REGION Network 16: 100 - return - wait for handshake with other instances
   RUNG wire#powerrail
      { S7_Templates := "SrcType := Int" } EQ_Contact(in1 := #cnt, in2 := 100)
      wire#w1
      Move(in := 0.0, out1 => #HydraulicCylinder.PressureCmd)
      Move(in := 0.0, out1 => #HydraulicCylinder.FlowCmd)
   END_RUNG
   RUNG wire#w1
      R_Coil( #dataDigiforce.Start )
   END_RUNG
   RUNG wire#w1
      Coil( #dataFitting.Returning )
   END_RUNG
   RUNG wire#w1
      Contact( #dataFitting.ContinueReturn )
      Move(in := 105, out1 => #cnt)
   END_RUNG
   // the same network as SCL:
   #_w1 := #cnt = 100;
   IF #_w1 THEN
       #HydraulicCylinder.PressureCmd := 0.0;
       #HydraulicCylinder.FlowCmd := 0.0;
       #dataDigiforce.Start := FALSE;
   END_IF;
   #dataFitting.Returning := #_w1;
   IF #_w1 AND #dataFitting.ContinueReturn THEN #cnt := 105; END_IF;
END_REGION

REGION Network 17: 105 - Start returning
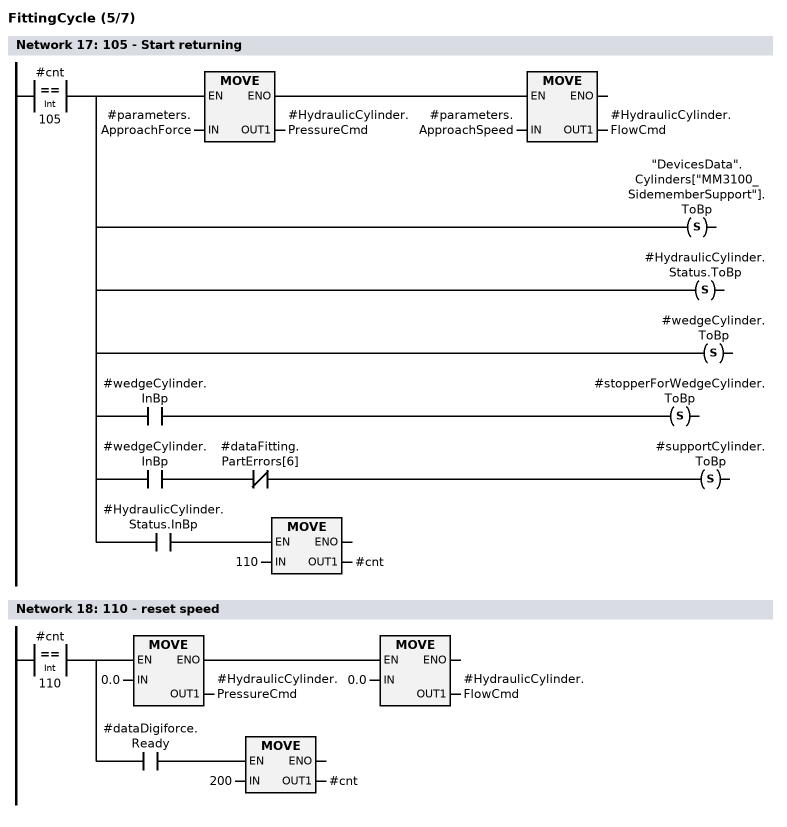
   RUNG wire#powerrail
      { S7_Templates := "SrcType := Int" } EQ_Contact(in1 := #cnt, in2 := 105)
      wire#w1
      Move(in := #parameters.ApproachForce, out1 => #HydraulicCylinder.PressureCmd)
      Move(in := #parameters.ApproachSpeed, out1 => #HydraulicCylinder.FlowCmd)
   END_RUNG
   RUNG wire#w1
      S_Coil( "DevicesData".Cylinders["MM3100_SidememberSupport"].ToBp )
   END_RUNG
   RUNG wire#w1
      S_Coil( #HydraulicCylinder.Status.ToBp )
   END_RUNG
   RUNG wire#w1
      S_Coil( #wedgeCylinder.ToBp )
   END_RUNG
   RUNG wire#w1
      Contact( #wedgeCylinder.InBp )
      S_Coil( #stopperForWedgeCylinder.ToBp )
   END_RUNG
   RUNG wire#w1
      Contact( #wedgeCylinder.InBp )
      I_Contact( #dataFitting.PartErrors[6] )
      S_Coil( #supportCylinder.ToBp )
   END_RUNG
   RUNG wire#w1
      Contact( #HydraulicCylinder.Status.InBp )
      Move(in := 110, out1 => #cnt)
   END_RUNG
   // the same network as SCL:
   #_w1 := #cnt = 105;
   IF #_w1 THEN
       #HydraulicCylinder.PressureCmd := #parameters.ApproachForce;
       #HydraulicCylinder.FlowCmd := #parameters.ApproachSpeed;
       "DevicesData".Cylinders["MM3100_SidememberSupport"].ToBp := TRUE;
       #HydraulicCylinder.Status.ToBp := TRUE;
       #wedgeCylinder.ToBp := TRUE;
   END_IF;
   IF #_w1 AND #wedgeCylinder.InBp THEN #stopperForWedgeCylinder.ToBp := TRUE; END_IF;
   IF #_w1 AND #wedgeCylinder.InBp AND NOT #dataFitting.PartErrors[6] THEN
       #supportCylinder.ToBp := TRUE;
   END_IF;
   IF #_w1 AND #HydraulicCylinder.Status.InBp THEN #cnt := 110; END_IF;
END_REGION

REGION Network 18: 110 - reset speed
   RUNG wire#powerrail
      { S7_Templates := "SrcType := Int" } EQ_Contact(in1 := #cnt, in2 := 110)
      wire#w1
      Move(in := 0.0, out1 => #HydraulicCylinder.PressureCmd)
      Move(in := 0.0, out1 => #HydraulicCylinder.FlowCmd)
   END_RUNG
   RUNG wire#w1
      Contact( #dataDigiforce.Ready )
      Move(in := 200, out1 => #cnt)
   END_RUNG
   // the same network as SCL:
   #_w1 := #cnt = 110;
   IF #_w1 THEN
       #HydraulicCylinder.PressureCmd := 0.0;
       #HydraulicCylinder.FlowCmd := 0.0;
   END_IF;
   IF #_w1 AND #dataDigiforce.Ready THEN #cnt := 200; END_IF;
END_REGION

REGION Network 19: 200 - Move all cylinders to basic - evaluate result
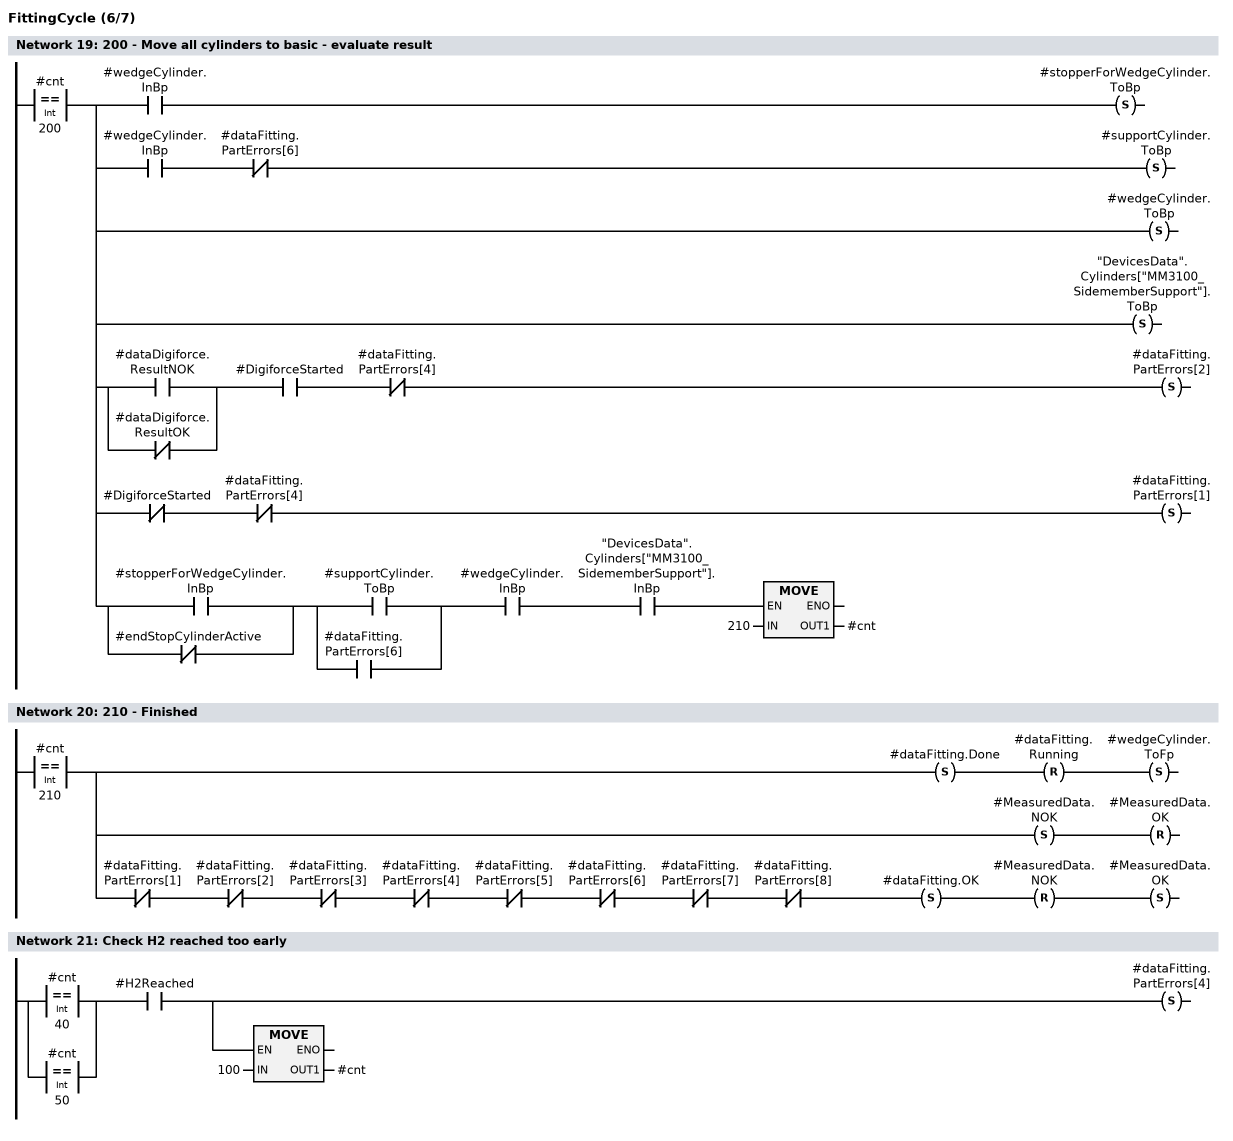
   RUNG wire#powerrail
      { S7_Templates := "SrcType := Int" } EQ_Contact(in1 := #cnt, in2 := 200)
      wire#w1
      Contact( #wedgeCylinder.InBp )
      S_Coil( #stopperForWedgeCylinder.ToBp )
   END_RUNG
   RUNG wire#w1
      Contact( #wedgeCylinder.InBp )
      I_Contact( #dataFitting.PartErrors[6] )
      S_Coil( #supportCylinder.ToBp )
   END_RUNG
   RUNG wire#w1
      S_Coil( #wedgeCylinder.ToBp )
   END_RUNG
   RUNG wire#w1
      S_Coil( "DevicesData".Cylinders["MM3100_SidememberSupport"].ToBp )
   END_RUNG
   RUNG wire#w1
      Contact( #dataDigiforce.ResultNOK )
      wire#w2
      Contact( #DigiforceStarted )
      I_Contact( #dataFitting.PartErrors[4] )
      S_Coil( #dataFitting.PartErrors[2] )
   END_RUNG
   RUNG wire#w1
      I_Contact( #dataDigiforce.ResultOK )
   END_RUNG wire#w2
   RUNG wire#w1
      I_Contact( #DigiforceStarted )
      I_Contact( #dataFitting.PartErrors[4] )
      S_Coil( #dataFitting.PartErrors[1] )
   END_RUNG
   RUNG wire#w1
      Contact( #stopperForWedgeCylinder.InBp )
      wire#w3
      Contact( #supportCylinder.ToBp )
      wire#w4
      Contact( #wedgeCylinder.InBp )
      Contact( "DevicesData".Cylinders["MM3100_SidememberSupport"].InBp )
      Move(in := 210, out1 => #cnt)
   END_RUNG
   RUNG wire#w1
      I_Contact( #endStopCylinderActive )
   END_RUNG wire#w3
   RUNG wire#w3
      Contact( #dataFitting.PartErrors[6] )
   END_RUNG wire#w4
   // the same network as SCL:
   #_w1 := #cnt = 200;
   IF #_w1 AND #wedgeCylinder.InBp THEN #stopperForWedgeCylinder.ToBp := TRUE; END_IF;
   IF #_w1 AND #wedgeCylinder.InBp AND NOT #dataFitting.PartErrors[6] THEN
       #supportCylinder.ToBp := TRUE;
   END_IF;
   IF #_w1 THEN
       #wedgeCylinder.ToBp := TRUE;
       "DevicesData".Cylinders["MM3100_SidememberSupport"].ToBp := TRUE;
   END_IF;
   IF #_w1 AND (#dataDigiforce.ResultNOK OR NOT #dataDigiforce.ResultOK) AND #DigiforceStarted AND NOT #dataFitting.PartErrors[4] THEN
       #dataFitting.PartErrors[2] := TRUE;
   END_IF;
   IF #_w1 AND NOT #DigiforceStarted AND NOT #dataFitting.PartErrors[4] THEN
       #dataFitting.PartErrors[1] := TRUE;
   END_IF;
   IF #_w1 AND (#stopperForWedgeCylinder.InBp OR NOT #endStopCylinderActive) AND (#supportCylinder.ToBp OR #dataFitting.PartErrors[6]) AND #wedgeCylinder.InBp AND "DevicesData".Cylinders["MM3100_SidememberSupport"].InBp THEN
       #cnt := 210;
   END_IF;
END_REGION

REGION Network 20: 210 - Finished
   RUNG wire#powerrail
      { S7_Templates := "SrcType := Int" } EQ_Contact(in1 := #cnt, in2 := 210)
      wire#w1
      S_Coil( #dataFitting.Done )
      R_Coil( #dataFitting.Running )
      S_Coil( #wedgeCylinder.ToFp )
   END_RUNG
   RUNG wire#w1
      S_Coil( #MeasuredData.NOK )
      R_Coil( #MeasuredData.OK )
   END_RUNG
   RUNG wire#w1
      I_Contact( #dataFitting.PartErrors[1] )
      I_Contact( #dataFitting.PartErrors[2] )
      I_Contact( #dataFitting.PartErrors[3] )
      I_Contact( #dataFitting.PartErrors[4] )
      I_Contact( #dataFitting.PartErrors[5] )
      I_Contact( #dataFitting.PartErrors[6] )
      I_Contact( #dataFitting.PartErrors[7] )
      I_Contact( #dataFitting.PartErrors[8] )
      S_Coil( #dataFitting.OK )
      R_Coil( #MeasuredData.NOK )
      S_Coil( #MeasuredData.OK )
   END_RUNG
   // the same network as SCL:
   #_w1 := #cnt = 210;
   IF #_w1 THEN
       #dataFitting.Done := TRUE;
       #dataFitting.Running := FALSE;
       #wedgeCylinder.ToFp := TRUE;
       #MeasuredData.NOK := TRUE;
       #MeasuredData.OK := FALSE;
   END_IF;
   IF #_w1 AND NOT #dataFitting.PartErrors[1] AND NOT #dataFitting.PartErrors[2] AND NOT #dataFitting.PartErrors[3] AND NOT #dataFitting.PartErrors[4] AND NOT #dataFitting.PartErrors[5] AND NOT #dataFitting.PartErrors[6] AND NOT #dataFitting.PartErrors[7] AND NOT #dataFitting.PartErrors[8] THEN
       #dataFitting.OK := TRUE;
       #MeasuredData.NOK := FALSE;
       #MeasuredData.OK := TRUE;
   END_IF;
END_REGION

REGION Network 21: Check H2 reached too early
   RUNG wire#powerrail
      { S7_Templates := "SrcType := Int" } EQ_Contact(in1 := #cnt, in2 := 40)
      wire#w1
      Contact( #H2Reached )
      wire#w2
      S_Coil( #dataFitting.PartErrors[4] )
   END_RUNG
   RUNG wire#powerrail
      { S7_Templates := "SrcType := Int" } EQ_Contact(in1 := #cnt, in2 := 50)
   END_RUNG wire#w1
   RUNG wire#w2
      Move(in := 100, out1 => #cnt)
   END_RUNG
   // the same network as SCL:
   IF ((#cnt = 40) OR (#cnt = 50)) AND #H2Reached THEN
       #dataFitting.PartErrors[4] := TRUE;
       #cnt := 100;
   END_IF;
END_REGION

REGION Network 22: Timeout
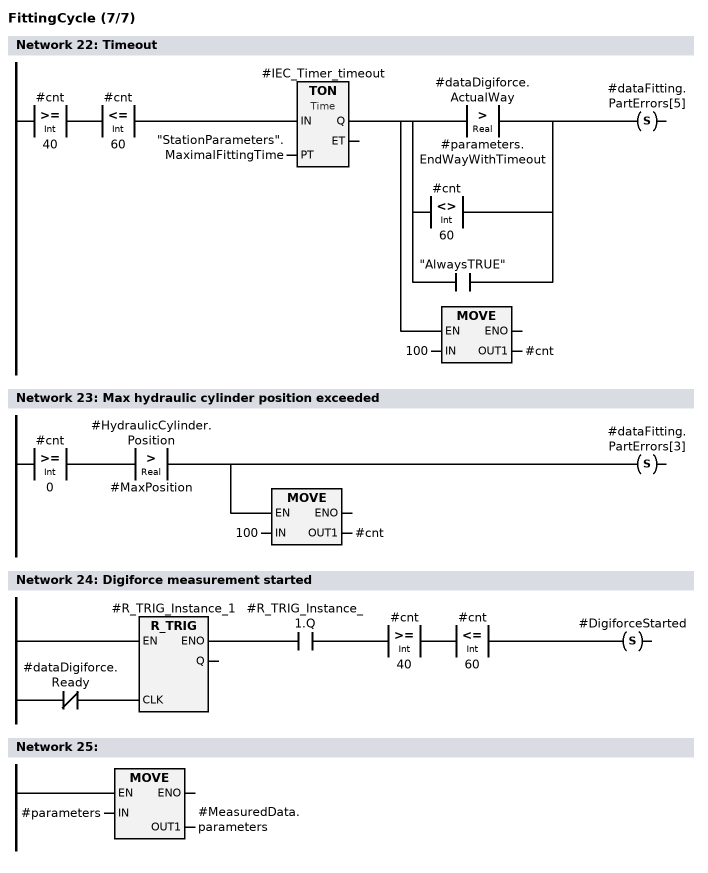
   RUNG wire#powerrail
      { S7_Templates := "SrcType := Int" } GE_Contact(in1 := #cnt, in2 := 40)
      { S7_Templates := "SrcType := Int" } LE_Contact(in1 := #cnt, in2 := 60)
      { S7_Templates := "time_type := Time" } #IEC_Timer_timeout.TON(pt := "StationParameters".MaximalFittingTime, et =>)
      wire#w1
      { S7_Templates := "SrcType := Real" } GT_Contact(in1 := #dataDigiforce.ActualWay, in2 := #parameters.EndWayWithTimeout)
      wire#w2
      S_Coil( #dataFitting.PartErrors[5] )
   END_RUNG
   RUNG wire#w1
      { S7_Templates := "SrcType := Int" } NE_Contact(in1 := #cnt, in2 := 60)
   END_RUNG wire#w2
   RUNG wire#w1
      Contact( "AlwaysTRUE" )
   END_RUNG wire#w2
   RUNG wire#w1
      Move(in := 100, out1 => #cnt)
   END_RUNG
   // the same network as SCL:
   #IEC_Timer_timeout(IN := (#cnt >= 40) AND (#cnt <= 60), PT := "StationParameters".MaximalFittingTime);   // TON
   IF #IEC_Timer_timeout.Q AND ((#dataDigiforce.ActualWay > #parameters.EndWayWithTimeout) OR (#cnt <> 60) OR "AlwaysTRUE") THEN
       #dataFitting.PartErrors[5] := TRUE;
   END_IF;
   IF #IEC_Timer_timeout.Q THEN #cnt := 100; END_IF;
END_REGION

REGION Network 23: Max hydraulic cylinder position exceeded
   RUNG wire#powerrail
      { S7_Templates := "SrcType := Int" } GE_Contact(in1 := #cnt, in2 := 0)
      { S7_Templates := "SrcType := Real" } GT_Contact(in1 := #HydraulicCylinder.Position, in2 := #MaxPosition)
      wire#w1
      S_Coil( #dataFitting.PartErrors[3] )
   END_RUNG
   RUNG wire#w1
      Move(in := 100, out1 => #cnt)
   END_RUNG
   // the same network as SCL:
   IF (#cnt >= 0) AND (#HydraulicCylinder.Position > #MaxPosition) THEN
       #dataFitting.PartErrors[3] := TRUE;
       #cnt := 100;
   END_IF;
END_REGION

REGION Network 24: Digiforce measurement started
   RUNG wire#powerrail
      #R_TRIG_Instance_1.R_TRIG(CLK := wire#w1, Q =>)
      Contact( #R_TRIG_Instance_1.Q )
      { S7_Templates := "SrcType := Int" } GE_Contact(in1 := #cnt, in2 := 40)
      { S7_Templates := "SrcType := Int" } LE_Contact(in1 := #cnt, in2 := 60)
      S_Coil( #DigiforceStarted )
   END_RUNG
   RUNG wire#powerrail
      I_Contact( #dataDigiforce.Ready )
   END_RUNG wire#w1
   // the same network as SCL:
   #R_TRIG_Instance_1(CLK := NOT #dataDigiforce.Ready, ENO => #_w1);   // R_TRIG
   IF #_w1 AND #R_TRIG_Instance_1.Q AND (#cnt >= 40) AND (#cnt <= 60) THEN #DigiforceStarted := TRUE; END_IF;
END_REGION

REGION Network 25
   RUNG wire#powerrail
      Move(in := #parameters, out1 => #MeasuredData.parameters)
   END_RUNG
   // the same network as SCL:
   #MeasuredData.parameters := #parameters;
END_REGION
END_FUNCTION_BLOCK

FUNCTION_BLOCK "HydraulicCylinder"   // FB17, LAD
{ S7_Optimized_Access := 'TRUE' }
VERSION : 0.1
// stored: AutoNumber true, IsIECCheckEnabled false, IsRetainMemResEnabled false, MemoryReserve 100, SetENOAutomatically false, UDAEnableTagReadback false
   VAR_INPUT
      HydraulicActive : Bool;
      BasicPositionMin : Real;
      BasicPositionMax : Real;
      MaxPosition : Real;
      ManualCommand : Int;
      CylinderNumber : Int;
   END_VAR
   VAR_IN_OUT
      data : "UDT_HydraulicCylinderData";
   END_VAR
   VAR
      dataOld : "UDT_HydraulicCylinderData";
      noCollision { S7_SetPoint := 'True'} : Bool;
      IEC_Timer_0_Instance { S7_SetPoint := 'True'} : TON_TIME;
      R_TRIG_Instance { S7_SetPoint := 'True'} : R_TRIG;
      difference { S7_SetPoint := 'True'} : Real;
      re : Real;
      IEC_Timer_0_Instance_1 { S7_SetPoint := 'True'} : TON_TIME;
      RampFunction_Instance { S7_SetPoint := 'True'} : RampFunction;
      BasicPositionMin_1mm_margin : Real;
      BasicPositionMax_1mm_margin : Real;
   END_VAR
   VAR_TEMP
      command : Int;
   END_VAR
   VAR_TEMP   // added for the SCL form of the ladder/FBD networks
      _w1 : Bool;
   END_VAR
BEGIN

REGION Network 1
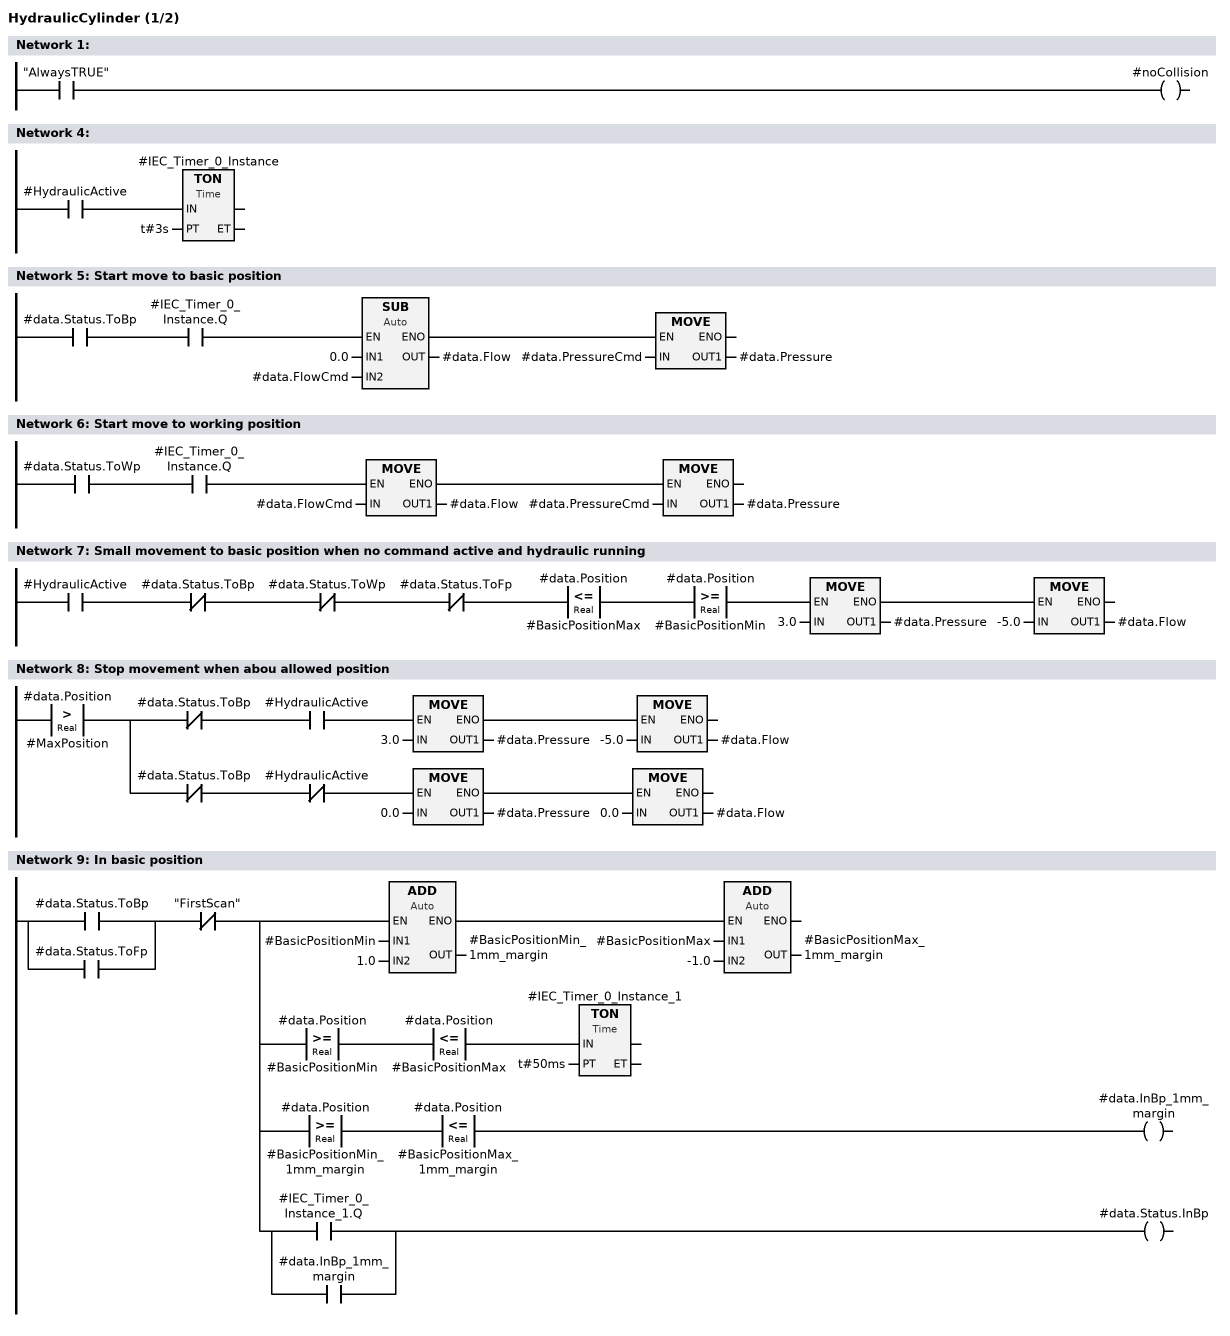
   RUNG wire#powerrail
      Contact( "AlwaysTRUE" )
      Coil( #noCollision )
   END_RUNG
   // the same network as SCL:
   #noCollision := "AlwaysTRUE";
END_REGION

REGION Network 2 (SCL)
   #command := #ManualCommand - #CylinderNumber;

   IF #command > 100 THEN
       "SandBoxData".MnualCommandMem := #command;
   END_IF;
   IF #command = 5000 THEN
       #data.Status.ToBp := true;
   END_IF;
   IF #command = 6000 THEN
       #data.Status.ToWp := true;
   END_IF;
   IF #command = 7000 THEN
       #data.Status.ToFp := true;
   END_IF;
END_REGION

REGION Network 3 (SCL): check new cylinder command
   //check if basic position req movement changed
   IF #data.Status.ToBp <> #dataOld.Status.ToBp AND #data.Status.ToBp THEN
       #data.Status.ToFp := false;
       #data.Status.ToWp := false;
       IF #noCollision THEN
           #data.Status.ToFp := false;
           #data.Status.ToWp := false;
       ELSE
           #data.Status.ToBp := false;
       END_IF;
   END_IF;
   //check if work position req movement changed
   IF #data.Status.ToWp <> #dataOld.Status.ToWp AND #data.Status.ToWp THEN
       IF #noCollision  THEN
           #data.Status.ToFp := false;
           #data.Status.ToBp := false;
       ELSE
           #data.Status.ToWp := false;
       END_IF;
   END_IF;
   //check if free position req movement changed
   IF #data.Status.ToFp <> #dataOld.Status.ToFp AND #data.Status.ToFp THEN
       #data.Status.ToBp := false;
       #data.Status.ToWp := false;
       IF #noCollision THEN
           #data.Status.ToBp := false;
           #data.Status.ToWp := false;
       ELSE
           #data.Status.ToFp := false;
       END_IF;
   END_IF;
   //store actual cylinder status to old
   #dataOld.Status := #data.Status;
END_REGION

REGION Network 4
   RUNG wire#powerrail
      Contact( #HydraulicActive )
      { S7_Templates := "time_type := Time" } #IEC_Timer_0_Instance.TON(pt := t#3s, et =>)
   END_RUNG
   // the same network as SCL:
   #IEC_Timer_0_Instance(IN := #HydraulicActive, PT := t#3s);   // TON
END_REGION

REGION Network 5: Start move to basic position
   RUNG wire#powerrail
      Contact( #data.Status.ToBp )
      Contact( #IEC_Timer_0_Instance.Q )
      Sub(in1 := 0.0, in2 := #data.FlowCmd, out => #data.Flow)
      Move(in := #data.PressureCmd, out1 => #data.Pressure)
   END_RUNG
   // the same network as SCL:
   IF #data.Status.ToBp AND #IEC_Timer_0_Instance.Q THEN
       #data.Flow := 0.0 - #data.FlowCmd;
       #data.Pressure := #data.PressureCmd;
   END_IF;
END_REGION

REGION Network 6: Start move to working position
   RUNG wire#powerrail
      Contact( #data.Status.ToWp )
      Contact( #IEC_Timer_0_Instance.Q )
      Move(in := #data.FlowCmd, out1 => #data.Flow)
      Move(in := #data.PressureCmd, out1 => #data.Pressure)
   END_RUNG
   // the same network as SCL:
   IF #data.Status.ToWp AND #IEC_Timer_0_Instance.Q THEN
       #data.Flow := #data.FlowCmd;
       #data.Pressure := #data.PressureCmd;
   END_IF;
END_REGION

REGION Network 7: Small movement to basic position when no command active and hydraulic running
   RUNG wire#powerrail
      Contact( #HydraulicActive )
      I_Contact( #data.Status.ToBp )
      I_Contact( #data.Status.ToWp )
      I_Contact( #data.Status.ToFp )
      { S7_Templates := "SrcType := Real" } LE_Contact(in1 := #data.Position, in2 := #BasicPositionMax)
      { S7_Templates := "SrcType := Real" } GE_Contact(in1 := #data.Position, in2 := #BasicPositionMin)
      Move(in := 3.0, out1 => #data.Pressure)
      Move(in := -5.0, out1 => #data.Flow)
   END_RUNG
   // the same network as SCL:
   IF #HydraulicActive AND NOT #data.Status.ToBp AND NOT #data.Status.ToWp AND NOT #data.Status.ToFp AND (#data.Position <= #BasicPositionMax) AND (#data.Position >= #BasicPositionMin) THEN
       #data.Pressure := 3.0;
       #data.Flow := -5.0;
   END_IF;
END_REGION

REGION Network 8: Stop movement when abou allowed position
   RUNG wire#powerrail
      { S7_Templates := "SrcType := Real" } GT_Contact(in1 := #data.Position, in2 := #MaxPosition)
      wire#w1
      I_Contact( #data.Status.ToBp )
      Contact( #HydraulicActive )
      Move(in := 3.0, out1 => #data.Pressure)
      Move(in := -5.0, out1 => #data.Flow)
   END_RUNG
   RUNG wire#w1
      I_Contact( #data.Status.ToBp )
      I_Contact( #HydraulicActive )
      Move(in := 0.0, out1 => #data.Pressure)
      Move(in := 0.0, out1 => #data.Flow)
   END_RUNG
   // the same network as SCL:
   #_w1 := #data.Position > #MaxPosition;
   IF #_w1 AND NOT #data.Status.ToBp AND #HydraulicActive THEN
       #data.Pressure := 3.0;
       #data.Flow := -5.0;
   END_IF;
   IF #_w1 AND NOT #data.Status.ToBp AND NOT #HydraulicActive THEN
       #data.Pressure := 0.0;
       #data.Flow := 0.0;
   END_IF;
END_REGION

REGION Network 9: In basic position
   RUNG wire#powerrail
      Contact( #data.Status.ToBp )
      wire#w1
      I_Contact( "FirstScan" )
      wire#w2
      Add(in1 := #BasicPositionMin, in2 := 1.0, out => #BasicPositionMin_1mm_margin)
      Add(in1 := #BasicPositionMax, in2 := -1.0, out => #BasicPositionMax_1mm_margin)
   END_RUNG
   RUNG wire#powerrail
      Contact( #data.Status.ToFp )
   END_RUNG wire#w1
   RUNG wire#w2
      { S7_Templates := "SrcType := Real" } GE_Contact(in1 := #data.Position, in2 := #BasicPositionMin)
      { S7_Templates := "SrcType := Real" } LE_Contact(in1 := #data.Position, in2 := #BasicPositionMax)
      { S7_Templates := "time_type := Time" } #IEC_Timer_0_Instance_1.TON(pt := t#50ms, et =>)
   END_RUNG
   RUNG wire#w2
      { S7_Templates := "SrcType := Real" } GE_Contact(in1 := #data.Position, in2 := #BasicPositionMin_1mm_margin)
      { S7_Templates := "SrcType := Real" } LE_Contact(in1 := #data.Position, in2 := #BasicPositionMax_1mm_margin)
      Coil( #data.InBp_1mm_margin )
   END_RUNG
   RUNG wire#w2
      Contact( #IEC_Timer_0_Instance_1.Q )
      wire#w3
      Coil( #data.Status.InBp )
   END_RUNG
   RUNG wire#w2
      Contact( #data.InBp_1mm_margin )
   END_RUNG wire#w3
   // the same network as SCL:
   #_w1 := (#data.Status.ToBp OR #data.Status.ToFp) AND NOT "FirstScan";
   IF #_w1 THEN
       #BasicPositionMin_1mm_margin := #BasicPositionMin + 1.0;
       #BasicPositionMax_1mm_margin := #BasicPositionMax + (-1.0);
   END_IF;
   #IEC_Timer_0_Instance_1(IN := #_w1 AND (#data.Position >= #BasicPositionMin) AND (#data.Position <= #BasicPositionMax),   // TON
                           PT := t#50ms);
   #data.InBp_1mm_margin := #_w1 AND (#data.Position >= #BasicPositionMin_1mm_margin) AND (#data.Position <= #BasicPositionMax_1mm_margin);
   #data.Status.InBp := #_w1 AND (#IEC_Timer_0_Instance_1.Q OR #data.InBp_1mm_margin);
END_REGION

REGION Network 10: Stand still - start stand still
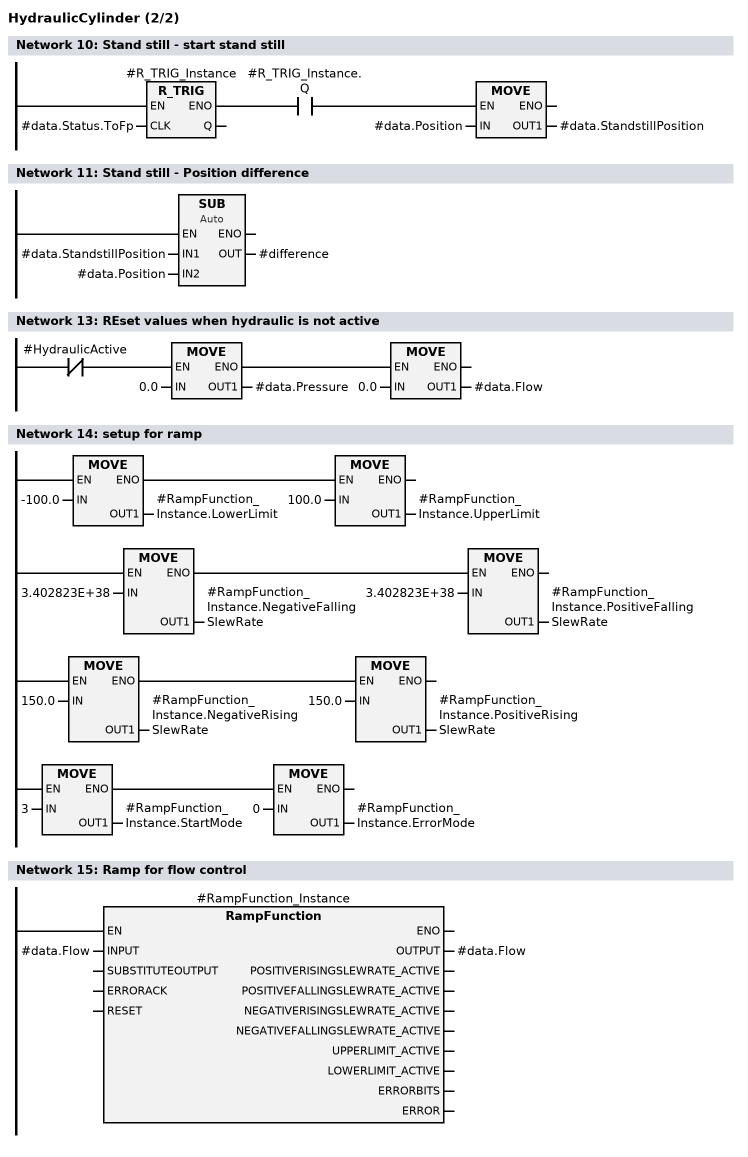
   RUNG wire#powerrail
      #R_TRIG_Instance.R_TRIG(CLK := #data.Status.ToFp, Q =>)
      Contact( #R_TRIG_Instance.Q )
      Move(in := #data.Position, out1 => #data.StandstillPosition)
   END_RUNG
   // the same network as SCL:
   #R_TRIG_Instance(CLK := #data.Status.ToFp, ENO => #_w1);   // R_TRIG
   IF #_w1 AND #R_TRIG_Instance.Q THEN #data.StandstillPosition := #data.Position; END_IF;
END_REGION

REGION Network 11: Stand still - Position difference
   RUNG wire#powerrail
      Sub(in1 := #data.StandstillPosition, in2 := #data.Position, out => #difference)
   END_RUNG
   // the same network as SCL:
   #difference := #data.StandstillPosition - #data.Position;
END_REGION

REGION Network 12 (SCL): Stand still - count regulation

   IF #data.Status.ToFp THEN
       #re := #difference;
       #re := #re * 10;
       IF #re > 0 THEN
           #re := #re + 5;
       END_IF;
       IF #re > 30 THEN
           #re := 30;
       END_IF;
       IF #re < -30 THEN
           #re := -30;
       END_IF;
       #data.Flow := #re;
       #data.Pressure := #data.PressureCmd;

       #data.Flow := 0;
       #data.Pressure := 0;

   END_IF;

   ;
END_REGION

REGION Network 13: REset values when hydraulic is not active
   RUNG wire#powerrail
      I_Contact( #HydraulicActive )
      Move(in := 0.0, out1 => #data.Pressure)
      Move(in := 0.0, out1 => #data.Flow)
   END_RUNG
   // the same network as SCL:
   IF NOT #HydraulicActive THEN
       #data.Pressure := 0.0;
       #data.Flow := 0.0;
   END_IF;
END_REGION

REGION Network 14: setup for ramp
   RUNG wire#powerrail
      Move(in := -100.0, out1 => #RampFunction_Instance.LowerLimit)
      Move(in := 100.0, out1 => #RampFunction_Instance.UpperLimit)
   END_RUNG
   RUNG wire#powerrail
      Move(in := 3.402823E+38, out1 => #RampFunction_Instance.NegativeFallingSlewRate)
      Move(in := 3.402823E+38, out1 => #RampFunction_Instance.PositiveFallingSlewRate)
   END_RUNG
   RUNG wire#powerrail
      Move(in := 150.0, out1 => #RampFunction_Instance.NegativeRisingSlewRate)
      Move(in := 150.0, out1 => #RampFunction_Instance.PositiveRisingSlewRate)
   END_RUNG
   RUNG wire#powerrail
      Move(in := 3, out1 => #RampFunction_Instance.StartMode)
      Move(in := 0, out1 => #RampFunction_Instance.ErrorMode)
   END_RUNG
   // the same network as SCL:
   #RampFunction_Instance.LowerLimit := -100.0;
   #RampFunction_Instance.UpperLimit := 100.0;
   #RampFunction_Instance.NegativeFallingSlewRate := 3.402823E+38;
   #RampFunction_Instance.PositiveFallingSlewRate := 3.402823E+38;
   #RampFunction_Instance.NegativeRisingSlewRate := 150.0;
   #RampFunction_Instance.PositiveRisingSlewRate := 150.0;
   #RampFunction_Instance.StartMode := 3;
   #RampFunction_Instance.ErrorMode := 0;
END_REGION

REGION Network 15: Ramp for flow control
   RUNG wire#powerrail
      #RampFunction_Instance.RampFunction(Input := #data.Flow, SubstituteOutput :=, ErrorAck :=, Reset :=, Output => #data.Flow, PositiveRisingSlewRate_Active =>, PositiveFallingSlewRate_Active =>, NegativeRisingSlewRate_Active =>, NegativeFallingSlewRate_Active =>, UpperLimit_Active =>, LowerLimit_Active =>, ErrorBits =>, Error =>)
   END_RUNG
   // the same network as SCL:
   #RampFunction_Instance(Input := #data.Flow, Output => #data.Flow);   // RampFunction
END_REGION
END_FUNCTION_BLOCK

FUNCTION_BLOCK "HydraulicMotor"   // FB36, LAD
{ S7_Optimized_Access := 'TRUE' }
VERSION : 0.1
// stored: AutoNumber true, IsIECCheckEnabled false, IsRetainMemResEnabled false, MemoryReserve 100, SetENOAutomatically false, UDAEnableTagReadback false
   VAR_INPUT
      cycleActiveCupforming : Bool;
      cycleActiveRiveting : Bool;
      temp1nok : Bool;
      temp2nok : Bool;
   END_VAR
   VAR_IN_OUT
      data : "UDT_HydraulicPump";
      qKM20 : Bool;
      qMotor : Bool;
      qValveCupforming : Bool;
      qValveRiveting : Bool;
   END_VAR
   VAR
      R_TRIG_Instance { S7_SetPoint := 'True'} : R_TRIG;
      cnt { S7_SetPoint := 'True'} : Int;
      IEC_Timer_0_Instance { S7_SetPoint := 'True'} : TON_TIME;
      F_TRIG_Instance { S7_SetPoint := 'True'} : F_TRIG;
      IEC_Timer_0_Instance_1 { S7_SetPoint := 'True'} : TON_TIME;
   END_VAR
   VAR_TEMP   // added for the SCL form of the ladder/FBD networks
      _w1 : Bool;
   END_VAR
BEGIN

REGION Network 1: Start auto mode
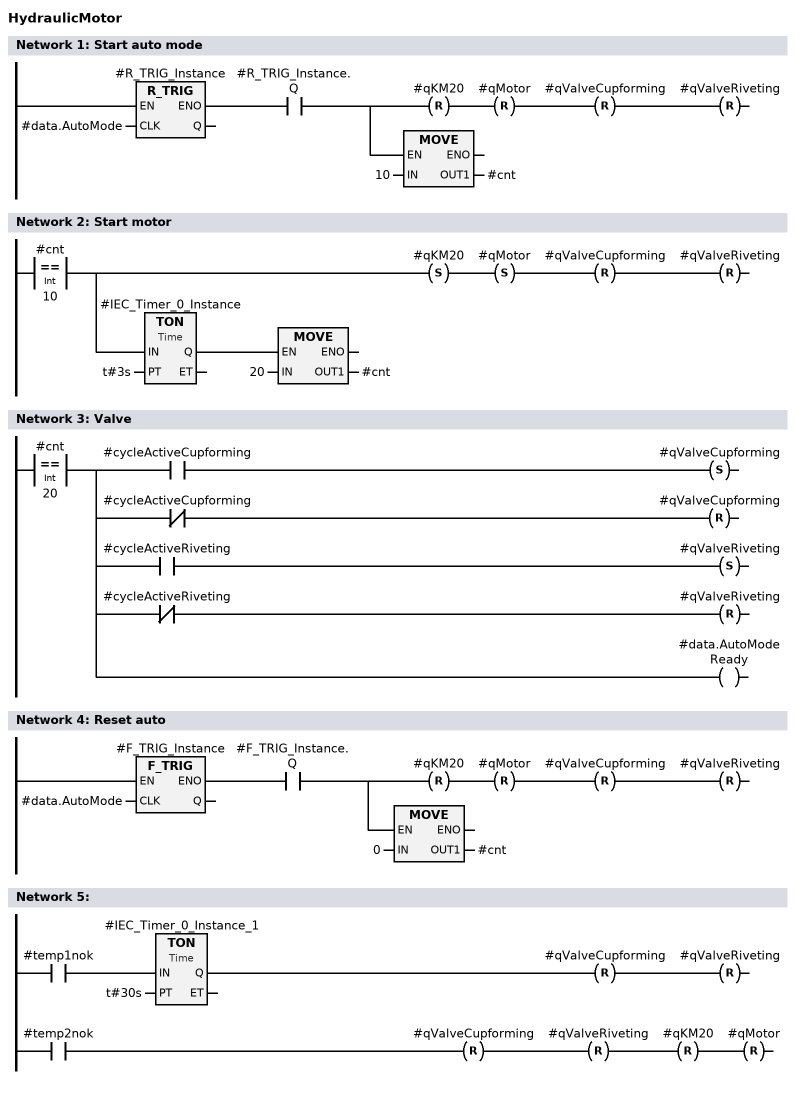
   RUNG wire#powerrail
      #R_TRIG_Instance.R_TRIG(CLK := #data.AutoMode, Q =>)
      Contact( #R_TRIG_Instance.Q )
      wire#w1
      R_Coil( #qKM20 )
      R_Coil( #qMotor )
      R_Coil( #qValveCupforming )
      R_Coil( #qValveRiveting )
   END_RUNG
   RUNG wire#w1
      Move(in := 10, out1 => #cnt)
   END_RUNG
   // the same network as SCL:
   #R_TRIG_Instance(CLK := #data.AutoMode, ENO => #_w1);   // R_TRIG
   IF #_w1 AND #R_TRIG_Instance.Q THEN
       #qKM20 := FALSE;
       #qMotor := FALSE;
       #qValveCupforming := FALSE;
       #qValveRiveting := FALSE;
       #cnt := 10;
   END_IF;
END_REGION

REGION Network 2: Start motor
   RUNG wire#powerrail
      { S7_Templates := "SrcType := Int" } EQ_Contact(in1 := #cnt, in2 := 10)
      wire#w1
      S_Coil( #qKM20 )
      S_Coil( #qMotor )
      R_Coil( #qValveCupforming )
      R_Coil( #qValveRiveting )
   END_RUNG
   RUNG wire#w1
      { S7_Templates := "time_type := Time" } #IEC_Timer_0_Instance.TON(pt := t#3s, et =>)
      Move(in := 20, out1 => #cnt)
   END_RUNG
   // the same network as SCL:
   #_w1 := #cnt = 10;
   IF #_w1 THEN
       #qKM20 := TRUE;
       #qMotor := TRUE;
       #qValveCupforming := FALSE;
       #qValveRiveting := FALSE;
   END_IF;
   #IEC_Timer_0_Instance(IN := #_w1, PT := t#3s);   // TON
   IF #IEC_Timer_0_Instance.Q THEN #cnt := 20; END_IF;
END_REGION

REGION Network 3: Valve
   RUNG wire#powerrail
      { S7_Templates := "SrcType := Int" } EQ_Contact(in1 := #cnt, in2 := 20)
      wire#w1
      Contact( #cycleActiveCupforming )
      S_Coil( #qValveCupforming )
   END_RUNG
   RUNG wire#w1
      I_Contact( #cycleActiveCupforming )
      R_Coil( #qValveCupforming )
   END_RUNG
   RUNG wire#w1
      Contact( #cycleActiveRiveting )
      S_Coil( #qValveRiveting )
   END_RUNG
   RUNG wire#w1
      I_Contact( #cycleActiveRiveting )
      R_Coil( #qValveRiveting )
   END_RUNG
   RUNG wire#w1
      Coil( #data.AutoModeReady )
   END_RUNG
   // the same network as SCL:
   #_w1 := #cnt = 20;
   IF #_w1 AND #cycleActiveCupforming THEN #qValveCupforming := TRUE; END_IF;
   IF #_w1 AND NOT #cycleActiveCupforming THEN #qValveCupforming := FALSE; END_IF;
   IF #_w1 AND #cycleActiveRiveting THEN #qValveRiveting := TRUE; END_IF;
   IF #_w1 AND NOT #cycleActiveRiveting THEN #qValveRiveting := FALSE; END_IF;
   #data.AutoModeReady := #_w1;
END_REGION

REGION Network 4: Reset auto
   RUNG wire#powerrail
      #F_TRIG_Instance.F_TRIG(CLK := #data.AutoMode, Q =>)
      Contact( #F_TRIG_Instance.Q )
      wire#w1
      R_Coil( #qKM20 )
      R_Coil( #qMotor )
      R_Coil( #qValveCupforming )
      R_Coil( #qValveRiveting )
   END_RUNG
   RUNG wire#w1
      Move(in := 0, out1 => #cnt)
   END_RUNG
   // the same network as SCL:
   #F_TRIG_Instance(CLK := #data.AutoMode, ENO => #_w1);   // F_TRIG
   IF #_w1 AND #F_TRIG_Instance.Q THEN
       #qKM20 := FALSE;
       #qMotor := FALSE;
       #qValveCupforming := FALSE;
       #qValveRiveting := FALSE;
       #cnt := 0;
   END_IF;
END_REGION

REGION Network 5
   RUNG wire#powerrail
      Contact( #temp1nok )
      { S7_Templates := "time_type := Time" } #IEC_Timer_0_Instance_1.TON(pt := t#30s, et =>)
      R_Coil( #qValveCupforming )
      R_Coil( #qValveRiveting )
   END_RUNG
   RUNG wire#powerrail
      Contact( #temp2nok )
      R_Coil( #qValveCupforming )
      R_Coil( #qValveRiveting )
      R_Coil( #qKM20 )
      R_Coil( #qMotor )
   END_RUNG
   // the same network as SCL:
   #IEC_Timer_0_Instance_1(IN := #temp1nok, PT := t#30s);   // TON
   IF #IEC_Timer_0_Instance_1.Q THEN
       #qValveCupforming := FALSE;
       #qValveRiveting := FALSE;
   END_IF;
   IF #temp2nok THEN
       #qValveCupforming := FALSE;
       #qValveRiveting := FALSE;
       #qKM20 := FALSE;
       #qMotor := FALSE;
   END_IF;
END_REGION
END_FUNCTION_BLOCK

FUNCTION_BLOCK "RobotControl"   // FB15, LAD
{ S7_Optimized_Access := 'TRUE' }
VERSION : 0.1
// stored: AutoNumber true, IsIECCheckEnabled false, IsRetainMemResEnabled false, MemoryReserve 100, SetENOAutomatically false, UDAEnableTagReadback false
   VAR_INPUT
      StartReq : Bool;
      KeyExt : Bool;
      JobNrReq : Byte;
      periReady : Bool;
      stopMess : Bool;
      progAct : Bool;
      onPath : Bool;
      ext : Bool;
      internalEstop : Bool;
      home : Bool;
      pgNoReq : Bool;
      robStopped : Bool;
      jobNrBack : Byte;
   END_VAR
   VAR_OUTPUT
      StartAllowed : Bool;
      Started : Bool;
      drivesOn : Bool;
      confMess : Bool;
      ExtStart : Bool;
      moveEnable : Bool;
      reqHome : Bool;
      pgNoValid : Bool;
      reqDoor : Bool;
      jobNr : Byte;
   END_VAR
BEGIN

REGION Network 1: Possible to start external auto
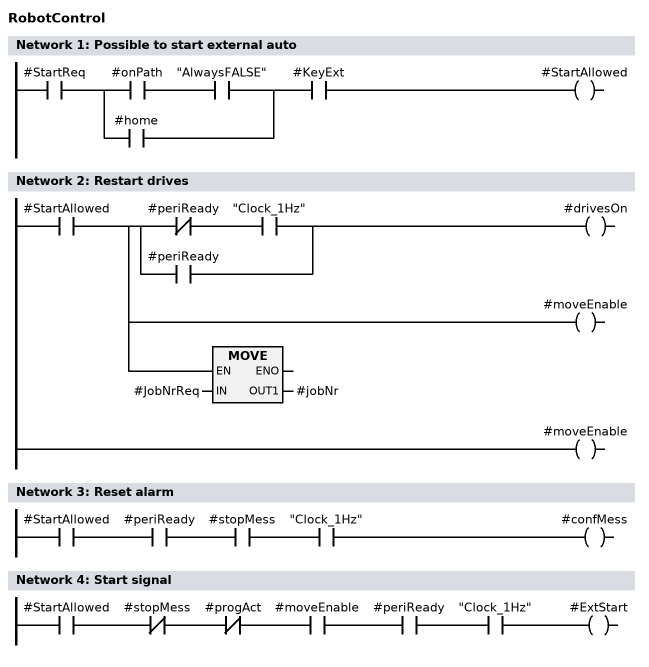
   RUNG wire#powerrail
      Contact( #StartReq )
      wire#w1
      Contact( #onPath )
      Contact( "AlwaysFALSE" )
      wire#w2
      Contact( #KeyExt )
      Coil( #StartAllowed )
   END_RUNG
   RUNG wire#w1
      Contact( #home )
   END_RUNG wire#w2
   // the same network as SCL:
   #StartAllowed := #StartReq AND ((#onPath AND "AlwaysFALSE") OR #home) AND #KeyExt;
END_REGION

REGION Network 2: Restart drives
   RUNG wire#powerrail
      Contact( #StartAllowed )
      wire#w1
      I_Contact( #periReady )
      Contact( "Clock_1Hz" )
      wire#w2
      Coil( #drivesOn )
   END_RUNG
   RUNG wire#w1
      Contact( #periReady )
   END_RUNG wire#w2
   RUNG wire#w1
      Coil( #moveEnable )
   END_RUNG
   RUNG wire#w1
      Move(in := #JobNrReq, out1 => #jobNr)
   END_RUNG
   RUNG wire#powerrail
      Coil( #moveEnable )
   END_RUNG
   // the same network as SCL:
   #drivesOn := #StartAllowed AND ((NOT #periReady AND "Clock_1Hz") OR #periReady);
   #moveEnable := #StartAllowed;
   IF #StartAllowed THEN #jobNr := #JobNrReq; END_IF;
   #moveEnable := TRUE;
END_REGION

REGION Network 3: Reset alarm
   RUNG wire#powerrail
      Contact( #StartAllowed )
      Contact( #periReady )
      Contact( #stopMess )
      Contact( "Clock_1Hz" )
      Coil( #confMess )
   END_RUNG
   // the same network as SCL:
   #confMess := #StartAllowed AND #periReady AND #stopMess AND "Clock_1Hz";
END_REGION

REGION Network 4: Start signal
   RUNG wire#powerrail
      Contact( #StartAllowed )
      I_Contact( #stopMess )
      I_Contact( #progAct )
      Contact( #moveEnable )
      Contact( #periReady )
      Contact( "Clock_1Hz" )
      Coil( #ExtStart )
   END_RUNG
   // the same network as SCL:
   #ExtStart := #StartAllowed AND NOT #stopMess AND NOT #progAct AND #moveEnable AND #periReady AND "Clock_1Hz";
END_REGION
END_FUNCTION_BLOCK

FUNCTION_BLOCK "RobotJob"   // FB45, GRAPH
VERSION : 0.1
// stored: AcknowledgeErrorsRequired true, AutoNumber true, GraphVersion 6.0, InitialValuesAcquisition false, IsIECCheckEnabled false, LanguageInNetworks LAD, LockOperatingMode false, PermanentILProcessingInMANMode false, SetENOAutomatically false, SkipSteps false, UDAEnableTagReadback false, WithAlarmHandling true
   // inherited from GRAPH_BASE
   VAR
      OFF_SQ_BASE : Bool;
   END_VAR
   VAR_INPUT
      OFF_SQ { ExternalAccessible := 'False'; ExternalVisible := 'False'; ExternalWritable := 'False'} : Bool := false;   // Turn sequence off
      INIT_SQ { ExternalAccessible := 'False'; ExternalVisible := 'False'; ExternalWritable := 'False'} : Bool := false;   // Set sequence to initial state
      ACK_EF { ExternalAccessible := 'False'; ExternalVisible := 'False'; ExternalWritable := 'False'} : Bool := false;   // Acknowledge all errors and faults
      S_PREV { ExternalAccessible := 'False'; ExternalVisible := 'False'; ExternalWritable := 'False'} : Bool := false;   // Output previous step in parameter S_NO
      S_NEXT { ExternalAccessible := 'False'; ExternalVisible := 'False'; ExternalWritable := 'False'} : Bool := false;   // Indicate next step in parameter S_NO
      SW_AUTO { ExternalAccessible := 'False'; ExternalVisible := 'False'; ExternalWritable := 'False'} : Bool := false;   // Automatic mode
      SW_TAP { ExternalAccessible := 'False'; ExternalVisible := 'False'; ExternalWritable := 'False'} : Bool := false;   // Semiautomatic/switch with transition
      SW_TOP { ExternalAccessible := 'False'; ExternalVisible := 'False'; ExternalWritable := 'False'} : Bool := false;   // Semiautomatic/ignore transition
      SW_MAN { ExternalAccessible := 'False'; ExternalVisible := 'False'; ExternalWritable := 'False'} : Bool := false;   // Manual mode
      S_SEL { ExternalAccessible := 'False'; ExternalVisible := 'False'; ExternalWritable := 'False'} : Int := 0;   // Select step to be output to S_NO
      S_ON { ExternalAccessible := 'False'; ExternalVisible := 'False'; ExternalWritable := 'False'} : Bool := false;   // Activate step indicated in S_NO
      S_OFF { ExternalAccessible := 'False'; ExternalVisible := 'False'; ExternalWritable := 'False'} : Bool := false;   // Deactivate step indicated S_NO
      T_PUSH { ExternalAccessible := 'False'; ExternalVisible := 'False'; ExternalWritable := 'False'} : Bool := false;   // Enable transition to switch in semi automatic mode
   END_VAR
   VAR_OUTPUT
      S_NO { ExternalAccessible := 'False'; ExternalVisible := 'False'; ExternalWritable := 'False'} : Int := 0;   // Step number
      S_MORE { ExternalAccessible := 'False'; ExternalVisible := 'False'; ExternalWritable := 'False'} : Bool := false;   // More steps are available and can be shown in S_NO
      S_ACTIVE { ExternalAccessible := 'False'; ExternalVisible := 'False'; ExternalWritable := 'False'} : Bool := false;   // Step indicated in S_NO is active
      ERR_FLT { ExternalAccessible := 'False'; ExternalVisible := 'False'; ExternalWritable := 'False'} : Bool := false;   // Interlock or supervision group error
      AUTO_ON { ExternalAccessible := 'False'; ExternalVisible := 'False'; ExternalWritable := 'False'} : Bool := false;   // Automatic mode is active
      TAP_ON { ExternalAccessible := 'False'; ExternalVisible := 'False'; ExternalWritable := 'False'} : Bool := false;   // Semiautomatic mode/step with transition enabled
      TOP_ON { ExternalAccessible := 'False'; ExternalVisible := 'False'; ExternalWritable := 'False'} : Bool := false;   // Semiautomatic mode/ignore transition enabled
      MAN_ON { ExternalAccessible := 'False'; ExternalVisible := 'False'; ExternalWritable := 'False'} : Bool := false;   // Manual mode is active
   END_VAR
BEGIN
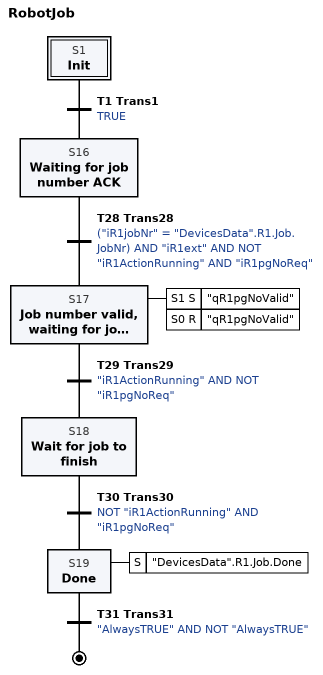
   // permanent pre-instructions
   NETWORK 1
      "DevicesData".R1.Job.Done := FALSE;

   // sequencer 1
   INITIAL_STEP Init:   // S1, max time T#10S, warning time T#7S
   END_STEP
   TRANSITION Trans1 FROM Init TO "Waiting for job number ACK"   // T1
      := TRUE;
   END_TRANSITION
   STEP "Waiting for job number ACK":   // S16, max time T#10S, warning time T#7S
      supervision V := #"Waiting for job number ACK".T > #"Waiting for job number ACK".T_MAX;
   END_STEP
   TRANSITION Trans28 FROM "Waiting for job number ACK" TO "Job number valid, waiting for job start"   // T28
      := ("iR1jobNr" = "DevicesData".R1.Job.JobNr) AND "iR1ext" AND NOT "iR1ActionRunning" AND "iR1pgNoReq";
   END_TRANSITION
   STEP "Job number valid, waiting for job start":   // S17, max time T#10S, warning time T#7S
      supervision V := #"Job number valid, waiting for job start".T > #"Job number valid, waiting for job start".T_MAX;
          S1  S    "qR1pgNoValid"
          S0  R    "qR1pgNoValid"
   END_STEP
   TRANSITION Trans29 FROM "Job number valid, waiting for job start" TO "Wait for job to finish"   // T29
      := "iR1ActionRunning" AND NOT "iR1pgNoReq";
   END_TRANSITION
   STEP "Wait for job to finish":   // S18, max time T#30S, warning time T#7S
      supervision V := #"Wait for job to finish".T > #"Wait for job to finish".T_MAX;
   END_STEP
   TRANSITION Trans30 FROM "Wait for job to finish" TO Done   // T30
      := NOT "iR1ActionRunning" AND "iR1pgNoReq";
   END_TRANSITION
   STEP Done:   // S19, max time T#10S, warning time T#7S
              S    "DevicesData".R1.Job.Done
   END_STEP
   TRANSITION Trans31 FROM Done TO END   // T31
      := "AlwaysTRUE" AND NOT "AlwaysTRUE";
   END_TRANSITION
END_FUNCTION_BLOCK

FUNCTION "READERS" : Void   // FC19, LAD
{ S7_Optimized_Access := 'TRUE' }
VERSION : 0.1
// stored: AutoNumber true, IsIECCheckEnabled false, SetENOAutomatically false, UDAEnableTagReadback false
   VAR_TEMP
      done1 : Bool;
      done2 : Bool;
      done3 : Bool;
      done4 : Bool;
      ERROR_RECIBIDO_ESCANER_REAR_TUBE : Int;
      ERROR_RECIBIDO_ESCANER_FRONT_TUBE : Int;
      ERROR_RECIBIDO_ESCANER_LH_MEMBER : Int;
      ERROR_RECIBIDO_ESCANER_RH_MEMBER : Int;
   END_VAR
   VAR_TEMP   // added for the SCL form of the ladder/FBD networks
      _w1 : Bool;
   END_VAR
BEGIN

REGION Network 1: INIT
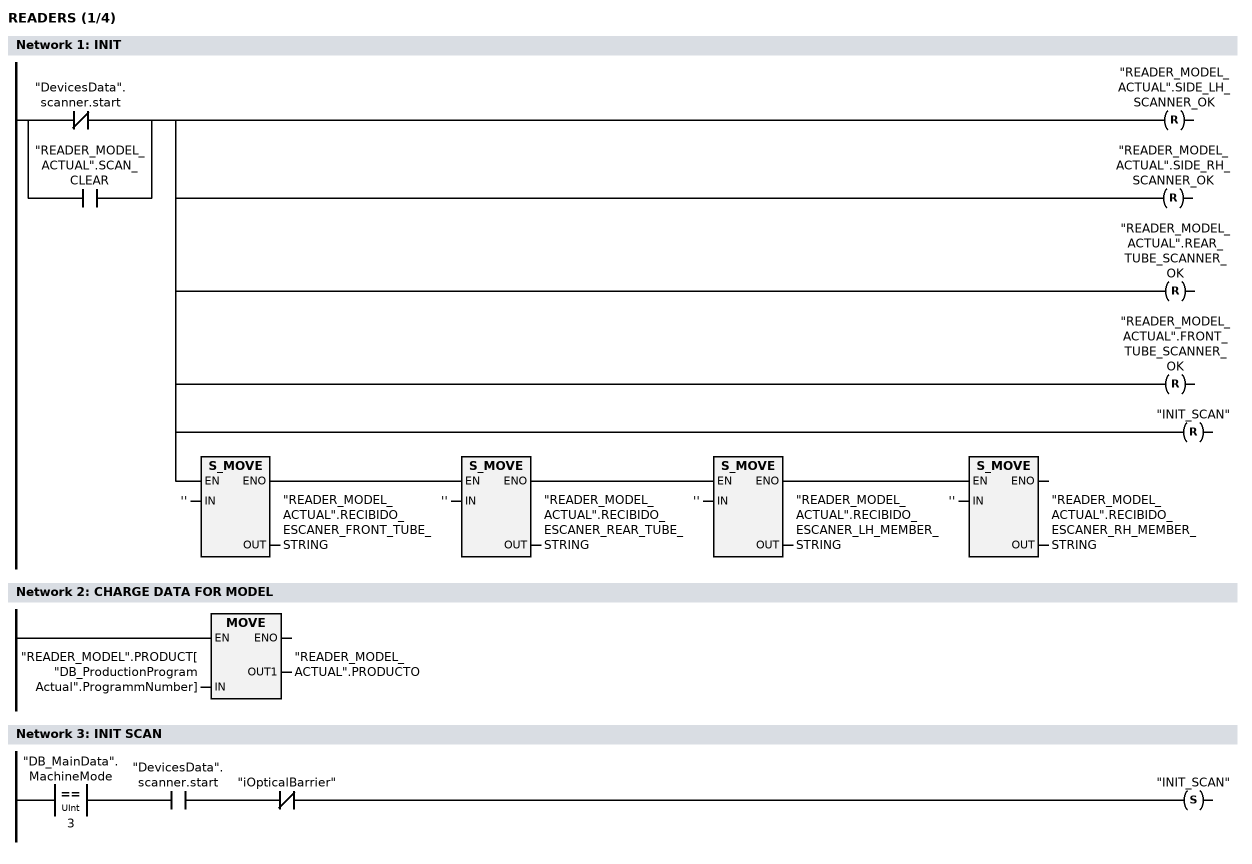
   RUNG wire#powerrail
      I_Contact( "DevicesData".scanner.start )
      wire#w1
      R_Coil( "READER_MODEL_ACTUAL".SIDE_LH_SCANNER_OK )
   END_RUNG
   RUNG wire#powerrail
      Contact( "READER_MODEL_ACTUAL".SCAN_CLEAR )
   END_RUNG wire#w1
   RUNG wire#w1
      R_Coil( "READER_MODEL_ACTUAL".SIDE_RH_SCANNER_OK )
   END_RUNG
   RUNG wire#w1
      R_Coil( "READER_MODEL_ACTUAL".REAR_TUBE_SCANNER_OK )
   END_RUNG
   RUNG wire#w1
      R_Coil( "READER_MODEL_ACTUAL".FRONT_TUBE_SCANNER_OK )
   END_RUNG
   RUNG wire#w1
      R_Coil( "INIT_SCAN" )
   END_RUNG
   RUNG wire#w1
      S_Move(in := '', out => "READER_MODEL_ACTUAL".RECIBIDO_ESCANER_FRONT_TUBE_STRING)
      S_Move(in := '', out => "READER_MODEL_ACTUAL".RECIBIDO_ESCANER_REAR_TUBE_STRING)
      S_Move(in := '', out => "READER_MODEL_ACTUAL".RECIBIDO_ESCANER_LH_MEMBER_STRING)
      S_Move(in := '', out => "READER_MODEL_ACTUAL".RECIBIDO_ESCANER_RH_MEMBER_STRING)
   END_RUNG
   // the same network as SCL:
   IF NOT "DevicesData".scanner.start OR "READER_MODEL_ACTUAL".SCAN_CLEAR THEN
       "READER_MODEL_ACTUAL".SIDE_LH_SCANNER_OK := FALSE;
       "READER_MODEL_ACTUAL".SIDE_RH_SCANNER_OK := FALSE;
       "READER_MODEL_ACTUAL".REAR_TUBE_SCANNER_OK := FALSE;
       "READER_MODEL_ACTUAL".FRONT_TUBE_SCANNER_OK := FALSE;
       "INIT_SCAN" := FALSE;
       "READER_MODEL_ACTUAL".RECIBIDO_ESCANER_FRONT_TUBE_STRING := '';
       "READER_MODEL_ACTUAL".RECIBIDO_ESCANER_REAR_TUBE_STRING := '';
       "READER_MODEL_ACTUAL".RECIBIDO_ESCANER_LH_MEMBER_STRING := '';
       "READER_MODEL_ACTUAL".RECIBIDO_ESCANER_RH_MEMBER_STRING := '';
   END_IF;
END_REGION

REGION Network 2: CHARGE DATA FOR MODEL
   RUNG wire#powerrail
      Move(in := "READER_MODEL".PRODUCT["DB_ProductionProgramActual".ProgrammNumber], out1 => "READER_MODEL_ACTUAL".PRODUCTO)
   END_RUNG
   // the same network as SCL:
   "READER_MODEL_ACTUAL".PRODUCTO := "READER_MODEL".PRODUCT["DB_ProductionProgramActual".ProgrammNumber];
END_REGION

REGION Network 3: INIT SCAN
   RUNG wire#powerrail
      { S7_Templates := "SrcType := UInt" } EQ_Contact(in1 := "DB_MainData".MachineMode, in2 := 3)
      Contact( "DevicesData".scanner.start )
      I_Contact( "iOpticalBarrier" )
      S_Coil( "INIT_SCAN" )
   END_RUNG
   // the same network as SCL:
   IF ("DB_MainData".MachineMode = 3) AND "DevicesData".scanner.start AND NOT "iOpticalBarrier" THEN
       "INIT_SCAN" := TRUE;
   END_IF;
END_REGION

REGION Network 4: LECTURA ESCANER REAR TUBE
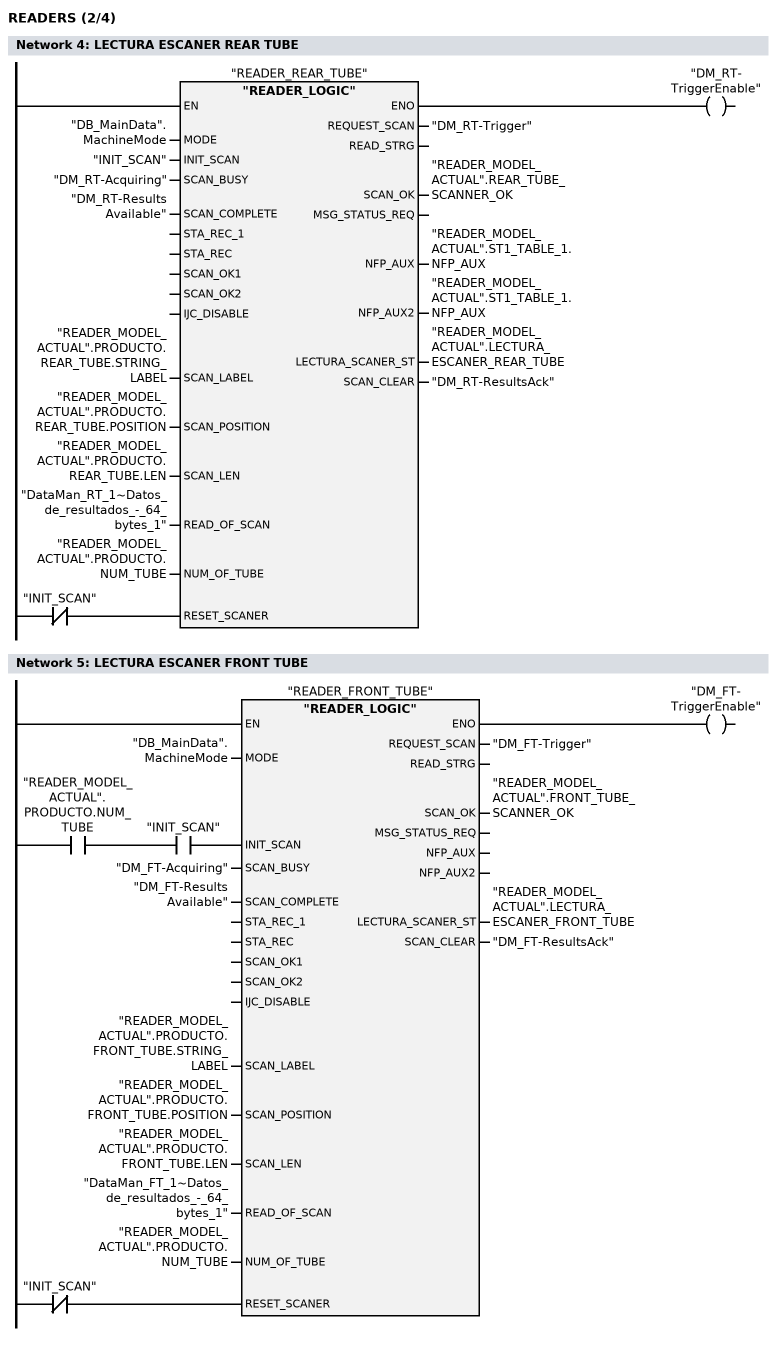
   RUNG wire#powerrail
      "READER_REAR_TUBE"(RESET_SCANER := wire#w1, MODE := "DB_MainData".MachineMode, INIT_SCAN := "INIT_SCAN", SCAN_BUSY := "DM_RT-Acquiring", SCAN_COMPLETE := "DM_RT-Results Available", STA_REC_1 :=, STA_REC :=, SCAN_OK1 :=, SCAN_OK2 :=, IJC_DISABLE :=, SCAN_LABEL := "READER_MODEL_ACTUAL".PRODUCTO.REAR_TUBE.STRING_LABEL, SCAN_POSITION := "READER_MODEL_ACTUAL".PRODUCTO.REAR_TUBE.POSITION, SCAN_LEN := "READER_MODEL_ACTUAL".PRODUCTO.REAR_TUBE.LEN, READ_OF_SCAN := "DataMan_RT_1~Datos_de_resultados_-_64_bytes_1", NUM_OF_TUBE := "READER_MODEL_ACTUAL".PRODUCTO.NUM_TUBE, REQUEST_SCAN => "DM_RT-Trigger", READ_STRG =>, SCAN_OK => "READER_MODEL_ACTUAL".REAR_TUBE_SCANNER_OK, MSG_STATUS_REQ =>, NFP_AUX => "READER_MODEL_ACTUAL".ST1_TABLE_1.NFP_AUX, NFP_AUX2 => "READER_MODEL_ACTUAL".ST1_TABLE_1.NFP_AUX, LECTURA_SCANER_ST => "READER_MODEL_ACTUAL".LECTURA_ESCANER_REAR_TUBE, SCAN_CLEAR => "DM_RT-ResultsAck")
      Coil( "DM_RT-TriggerEnable" )
   END_RUNG
   RUNG wire#powerrail
      I_Contact( "INIT_SCAN" )
   END_RUNG wire#w1
   // the same network as SCL:
   "READER_REAR_TUBE"(MODE := "DB_MainData".MachineMode,   // "READER_LOGIC"
                      INIT_SCAN := "INIT_SCAN",
                      SCAN_BUSY := "DM_RT-Acquiring",
                      SCAN_COMPLETE := "DM_RT-Results Available",
                      SCAN_LABEL := "READER_MODEL_ACTUAL".PRODUCTO.REAR_TUBE.STRING_LABEL,
                      SCAN_POSITION := "READER_MODEL_ACTUAL".PRODUCTO.REAR_TUBE.POSITION,
                      SCAN_LEN := "READER_MODEL_ACTUAL".PRODUCTO.REAR_TUBE.LEN,
                      READ_OF_SCAN := "DataMan_RT_1~Datos_de_resultados_-_64_bytes_1",
                      NUM_OF_TUBE := "READER_MODEL_ACTUAL".PRODUCTO.NUM_TUBE,
                      RESET_SCANER := NOT "INIT_SCAN",
                      REQUEST_SCAN => "DM_RT-Trigger",
                      SCAN_OK => "READER_MODEL_ACTUAL".REAR_TUBE_SCANNER_OK,
                      NFP_AUX => "READER_MODEL_ACTUAL".ST1_TABLE_1.NFP_AUX,
                      NFP_AUX2 => "READER_MODEL_ACTUAL".ST1_TABLE_1.NFP_AUX,
                      LECTURA_SCANER_ST => "READER_MODEL_ACTUAL".LECTURA_ESCANER_REAR_TUBE,
                      SCAN_CLEAR => "DM_RT-ResultsAck",
                      ENO => #_w1);
   "DM_RT-TriggerEnable" := #_w1;
END_REGION

REGION Network 5: LECTURA ESCANER FRONT TUBE
   RUNG wire#powerrail
      "READER_FRONT_TUBE"(INIT_SCAN := wire#w1, RESET_SCANER := wire#w2, MODE := "DB_MainData".MachineMode, SCAN_BUSY := "DM_FT-Acquiring", SCAN_COMPLETE := "DM_FT-Results Available", STA_REC_1 :=, STA_REC :=, SCAN_OK1 :=, SCAN_OK2 :=, IJC_DISABLE :=, SCAN_LABEL := "READER_MODEL_ACTUAL".PRODUCTO.FRONT_TUBE.STRING_LABEL, SCAN_POSITION := "READER_MODEL_ACTUAL".PRODUCTO.FRONT_TUBE.POSITION, SCAN_LEN := "READER_MODEL_ACTUAL".PRODUCTO.FRONT_TUBE.LEN, READ_OF_SCAN := "DataMan_FT_1~Datos_de_resultados_-_64_bytes_1", NUM_OF_TUBE := "READER_MODEL_ACTUAL".PRODUCTO.NUM_TUBE, REQUEST_SCAN => "DM_FT-Trigger", READ_STRG =>, SCAN_OK => "READER_MODEL_ACTUAL".FRONT_TUBE_SCANNER_OK, MSG_STATUS_REQ =>, NFP_AUX =>, NFP_AUX2 =>, LECTURA_SCANER_ST => "READER_MODEL_ACTUAL".LECTURA_ESCANER_FRONT_TUBE, SCAN_CLEAR => "DM_FT-ResultsAck")
      Coil( "DM_FT-TriggerEnable" )
   END_RUNG
   RUNG wire#powerrail
      Contact( "READER_MODEL_ACTUAL".PRODUCTO.NUM_TUBE )
      Contact( "INIT_SCAN" )
   END_RUNG wire#w1
   RUNG wire#powerrail
      I_Contact( "INIT_SCAN" )
   END_RUNG wire#w2
   // the same network as SCL:
   "READER_FRONT_TUBE"(MODE := "DB_MainData".MachineMode,   // "READER_LOGIC"
                       INIT_SCAN := "READER_MODEL_ACTUAL".PRODUCTO.NUM_TUBE AND "INIT_SCAN",
                       SCAN_BUSY := "DM_FT-Acquiring",
                       SCAN_COMPLETE := "DM_FT-Results Available",
                       SCAN_LABEL := "READER_MODEL_ACTUAL".PRODUCTO.FRONT_TUBE.STRING_LABEL,
                       SCAN_POSITION := "READER_MODEL_ACTUAL".PRODUCTO.FRONT_TUBE.POSITION,
                       SCAN_LEN := "READER_MODEL_ACTUAL".PRODUCTO.FRONT_TUBE.LEN,
                       READ_OF_SCAN := "DataMan_FT_1~Datos_de_resultados_-_64_bytes_1",
                       NUM_OF_TUBE := "READER_MODEL_ACTUAL".PRODUCTO.NUM_TUBE,
                       RESET_SCANER := NOT "INIT_SCAN",
                       REQUEST_SCAN => "DM_FT-Trigger",
                       SCAN_OK => "READER_MODEL_ACTUAL".FRONT_TUBE_SCANNER_OK,
                       LECTURA_SCANER_ST => "READER_MODEL_ACTUAL".LECTURA_ESCANER_FRONT_TUBE,
                       SCAN_CLEAR => "DM_FT-ResultsAck",
                       ENO => #_w1);
   "DM_FT-TriggerEnable" := #_w1;
END_REGION

REGION Network 6: LECTURA ESCANER SIDE LH
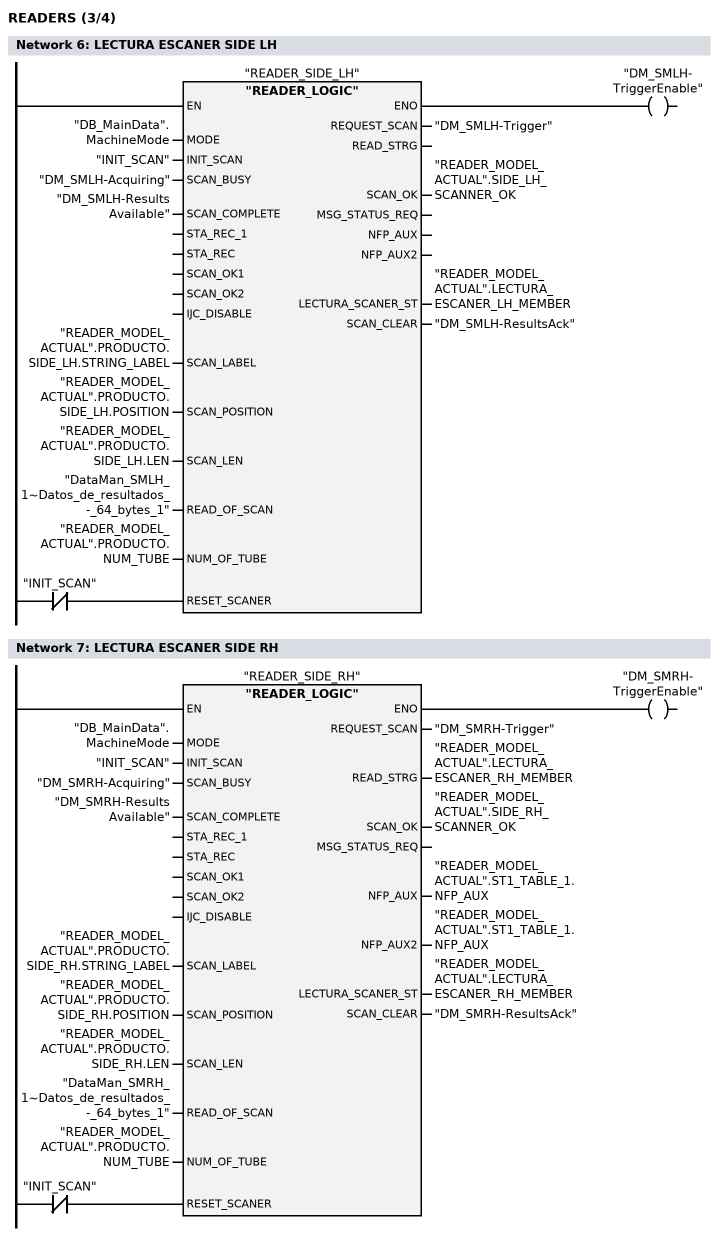
   RUNG wire#powerrail
      "READER_SIDE_LH"(RESET_SCANER := wire#w1, MODE := "DB_MainData".MachineMode, INIT_SCAN := "INIT_SCAN", SCAN_BUSY := "DM_SMLH-Acquiring", SCAN_COMPLETE := "DM_SMLH-Results Available", STA_REC_1 :=, STA_REC :=, SCAN_OK1 :=, SCAN_OK2 :=, IJC_DISABLE :=, SCAN_LABEL := "READER_MODEL_ACTUAL".PRODUCTO.SIDE_LH.STRING_LABEL, SCAN_POSITION := "READER_MODEL_ACTUAL".PRODUCTO.SIDE_LH.POSITION, SCAN_LEN := "READER_MODEL_ACTUAL".PRODUCTO.SIDE_LH.LEN, READ_OF_SCAN := "DataMan_SMLH_1~Datos_de_resultados_-_64_bytes_1", NUM_OF_TUBE := "READER_MODEL_ACTUAL".PRODUCTO.NUM_TUBE, REQUEST_SCAN => "DM_SMLH-Trigger", READ_STRG =>, SCAN_OK => "READER_MODEL_ACTUAL".SIDE_LH_SCANNER_OK, MSG_STATUS_REQ =>, NFP_AUX =>, NFP_AUX2 =>, LECTURA_SCANER_ST => "READER_MODEL_ACTUAL".LECTURA_ESCANER_LH_MEMBER, SCAN_CLEAR => "DM_SMLH-ResultsAck")
      Coil( "DM_SMLH-TriggerEnable" )
   END_RUNG
   RUNG wire#powerrail
      I_Contact( "INIT_SCAN" )
   END_RUNG wire#w1
   // the same network as SCL:
   "READER_SIDE_LH"(MODE := "DB_MainData".MachineMode,   // "READER_LOGIC"
                    INIT_SCAN := "INIT_SCAN",
                    SCAN_BUSY := "DM_SMLH-Acquiring",
                    SCAN_COMPLETE := "DM_SMLH-Results Available",
                    SCAN_LABEL := "READER_MODEL_ACTUAL".PRODUCTO.SIDE_LH.STRING_LABEL,
                    SCAN_POSITION := "READER_MODEL_ACTUAL".PRODUCTO.SIDE_LH.POSITION,
                    SCAN_LEN := "READER_MODEL_ACTUAL".PRODUCTO.SIDE_LH.LEN,
                    READ_OF_SCAN := "DataMan_SMLH_1~Datos_de_resultados_-_64_bytes_1",
                    NUM_OF_TUBE := "READER_MODEL_ACTUAL".PRODUCTO.NUM_TUBE,
                    RESET_SCANER := NOT "INIT_SCAN",
                    REQUEST_SCAN => "DM_SMLH-Trigger",
                    SCAN_OK => "READER_MODEL_ACTUAL".SIDE_LH_SCANNER_OK,
                    LECTURA_SCANER_ST => "READER_MODEL_ACTUAL".LECTURA_ESCANER_LH_MEMBER,
                    SCAN_CLEAR => "DM_SMLH-ResultsAck",
                    ENO => #_w1);
   "DM_SMLH-TriggerEnable" := #_w1;
END_REGION

REGION Network 7: LECTURA ESCANER SIDE RH
   RUNG wire#powerrail
      "READER_SIDE_RH"(RESET_SCANER := wire#w1, MODE := "DB_MainData".MachineMode, INIT_SCAN := "INIT_SCAN", SCAN_BUSY := "DM_SMRH-Acquiring", SCAN_COMPLETE := "DM_SMRH-Results Available", STA_REC_1 :=, STA_REC :=, SCAN_OK1 :=, SCAN_OK2 :=, IJC_DISABLE :=, SCAN_LABEL := "READER_MODEL_ACTUAL".PRODUCTO.SIDE_RH.STRING_LABEL, SCAN_POSITION := "READER_MODEL_ACTUAL".PRODUCTO.SIDE_RH.POSITION, SCAN_LEN := "READER_MODEL_ACTUAL".PRODUCTO.SIDE_RH.LEN, READ_OF_SCAN := "DataMan_SMRH_1~Datos_de_resultados_-_64_bytes_1", NUM_OF_TUBE := "READER_MODEL_ACTUAL".PRODUCTO.NUM_TUBE, REQUEST_SCAN => "DM_SMRH-Trigger", READ_STRG => "READER_MODEL_ACTUAL".LECTURA_ESCANER_RH_MEMBER, SCAN_OK => "READER_MODEL_ACTUAL".SIDE_RH_SCANNER_OK, MSG_STATUS_REQ =>, NFP_AUX => "READER_MODEL_ACTUAL".ST1_TABLE_1.NFP_AUX, NFP_AUX2 => "READER_MODEL_ACTUAL".ST1_TABLE_1.NFP_AUX, LECTURA_SCANER_ST => "READER_MODEL_ACTUAL".LECTURA_ESCANER_RH_MEMBER, SCAN_CLEAR => "DM_SMRH-ResultsAck")
      Coil( "DM_SMRH-TriggerEnable" )
   END_RUNG
   RUNG wire#powerrail
      I_Contact( "INIT_SCAN" )
   END_RUNG wire#w1
   // the same network as SCL:
   "READER_SIDE_RH"(MODE := "DB_MainData".MachineMode,   // "READER_LOGIC"
                    INIT_SCAN := "INIT_SCAN",
                    SCAN_BUSY := "DM_SMRH-Acquiring",
                    SCAN_COMPLETE := "DM_SMRH-Results Available",
                    SCAN_LABEL := "READER_MODEL_ACTUAL".PRODUCTO.SIDE_RH.STRING_LABEL,
                    SCAN_POSITION := "READER_MODEL_ACTUAL".PRODUCTO.SIDE_RH.POSITION,
                    SCAN_LEN := "READER_MODEL_ACTUAL".PRODUCTO.SIDE_RH.LEN,
                    READ_OF_SCAN := "DataMan_SMRH_1~Datos_de_resultados_-_64_bytes_1",
                    NUM_OF_TUBE := "READER_MODEL_ACTUAL".PRODUCTO.NUM_TUBE,
                    RESET_SCANER := NOT "INIT_SCAN",
                    REQUEST_SCAN => "DM_SMRH-Trigger",
                    READ_STRG => "READER_MODEL_ACTUAL".LECTURA_ESCANER_RH_MEMBER,
                    SCAN_OK => "READER_MODEL_ACTUAL".SIDE_RH_SCANNER_OK,
                    NFP_AUX => "READER_MODEL_ACTUAL".ST1_TABLE_1.NFP_AUX,
                    NFP_AUX2 => "READER_MODEL_ACTUAL".ST1_TABLE_1.NFP_AUX,
                    LECTURA_SCANER_ST => "READER_MODEL_ACTUAL".LECTURA_ESCANER_RH_MEMBER,
                    SCAN_CLEAR => "DM_SMRH-ResultsAck",
                    ENO => #_w1);
   "DM_SMRH-TriggerEnable" := #_w1;
END_REGION

REGION Network 8: ALL SCANER OK
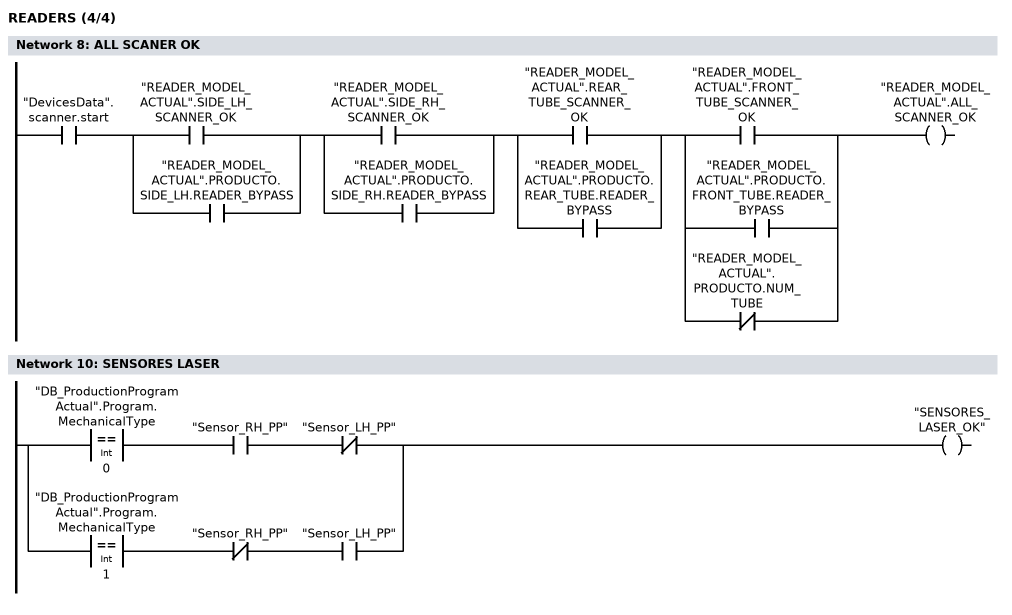
   RUNG wire#powerrail
      Contact( "DevicesData".scanner.start )
      wire#w1
      Contact( "READER_MODEL_ACTUAL".SIDE_LH_SCANNER_OK )
      wire#w2
      Contact( "READER_MODEL_ACTUAL".SIDE_RH_SCANNER_OK )
      wire#w3
      Contact( "READER_MODEL_ACTUAL".REAR_TUBE_SCANNER_OK )
      wire#w4
      Contact( "READER_MODEL_ACTUAL".FRONT_TUBE_SCANNER_OK )
      wire#w5
      Coil( "READER_MODEL_ACTUAL".ALL_SCANNER_OK )
   END_RUNG
   RUNG wire#w1
      Contact( "READER_MODEL_ACTUAL".PRODUCTO.SIDE_LH.READER_BYPASS )
   END_RUNG wire#w2
   RUNG wire#w2
      Contact( "READER_MODEL_ACTUAL".PRODUCTO.SIDE_RH.READER_BYPASS )
   END_RUNG wire#w3
   RUNG wire#w3
      Contact( "READER_MODEL_ACTUAL".PRODUCTO.REAR_TUBE.READER_BYPASS )
   END_RUNG wire#w4
   RUNG wire#w4
      Contact( "READER_MODEL_ACTUAL".PRODUCTO.FRONT_TUBE.READER_BYPASS )
   END_RUNG wire#w5
   RUNG wire#w4
      I_Contact( "READER_MODEL_ACTUAL".PRODUCTO.NUM_TUBE )
   END_RUNG wire#w5
   // the same network as SCL:
   "READER_MODEL_ACTUAL".ALL_SCANNER_OK := "DevicesData".scanner.start AND ("READER_MODEL_ACTUAL".SIDE_LH_SCANNER_OK OR "READER_MODEL_ACTUAL".PRODUCTO.SIDE_LH.READER_BYPASS) AND ("READER_MODEL_ACTUAL".SIDE_RH_SCANNER_OK OR "READER_MODEL_ACTUAL".PRODUCTO.SIDE_RH.READER_BYPASS) AND ("READER_MODEL_ACTUAL".REAR_TUBE_SCANNER_OK OR "READER_MODEL_ACTUAL".PRODUCTO.REAR_TUBE.READER_BYPASS) AND ("READER_MODEL_ACTUAL".FRONT_TUBE_SCANNER_OK OR "READER_MODEL_ACTUAL".PRODUCTO.FRONT_TUBE.READER_BYPASS OR NOT "READER_MODEL_ACTUAL".PRODUCTO.NUM_TUBE);
END_REGION

REGION Network 9: SEND TRC 1 MSG5
END_REGION

REGION Network 10: SENSORES LASER
   RUNG wire#powerrail
      { S7_Templates := "SrcType := Int" } EQ_Contact(in1 := "DB_ProductionProgramActual".Program.MechanicalType, in2 := 0)
      Contact( "Sensor_RH_PP" )
      I_Contact( "Sensor_LH_PP" )
      wire#w1
      Coil( "SENSORES_LASER_OK" )
   END_RUNG
   RUNG wire#powerrail
      { S7_Templates := "SrcType := Int" } EQ_Contact(in1 := "DB_ProductionProgramActual".Program.MechanicalType, in2 := 1)
      I_Contact( "Sensor_RH_PP" )
      Contact( "Sensor_LH_PP" )
   END_RUNG wire#w1
   // the same network as SCL:
   "SENSORES_LASER_OK" := (("DB_ProductionProgramActual".Program.MechanicalType = 0) AND "Sensor_RH_PP" AND NOT "Sensor_LH_PP") OR (("DB_ProductionProgramActual".Program.MechanicalType = 1) AND NOT "Sensor_RH_PP" AND "Sensor_LH_PP");
END_REGION
END_FUNCTION

FUNCTION_BLOCK "READER_LOGIC"   // FB24, LAD
{ S7_Optimized_Access := 'TRUE' }
VERSION : 0.1
// stored: AutoNumber true, IsIECCheckEnabled false, IsRetainMemResEnabled false, MemoryReserve 100, SetENOAutomatically false, UDAEnableTagReadback false
   VAR_INPUT
      MODE : UInt;
      INIT_SCAN : Bool;
      SCAN_BUSY : Bool;
      SCAN_COMPLETE : Bool;
      STA_REC_1 : Bool;
      STA_REC : Bool;
      SCAN_OK1 : Bool;
      SCAN_OK2 : Bool;
      IJC_DISABLE : Bool;
      SCAN_LABEL : String;
      SCAN_POSITION : Int;
      SCAN_LEN : Int;
      READ_OF_SCAN : HW_SUBMODULE;
      NUM_OF_TUBE : Bool;
      RESET_SCANER : Bool;
   END_VAR
   VAR_OUTPUT
      REQUEST_SCAN : Bool;
      READ_STRG : String;
      SCAN_OK : Bool;
      MSG_STATUS_REQ : Bool;
      NFP_AUX : String;
      NFP_AUX2 : String;
      LECTURA_SCANER_ST : String;
      SCAN_CLEAR : Bool;
   END_VAR
   VAR
      RET_TRIG : IEC_TIMER;
   END_VAR
   VAR_TEMP
      ERROR_RECIBIDO_ESCANER : Int;
      RECIBIDO_SCANER : Array[0..254] of Char;
      RECIBIDO_SCANER_STRG : String;
      LECTURA_SCANER : String;
      done : Bool;
   END_VAR
   VAR_TEMP   // added for the SCL form of the ladder/FBD networks
      _w1 : Bool;
      _w2 : Bool;
      _w3 : Bool;
      _w4 : Bool;
      _w5 : Bool;
      _w6 : Bool;
   END_VAR
BEGIN

REGION Network 1
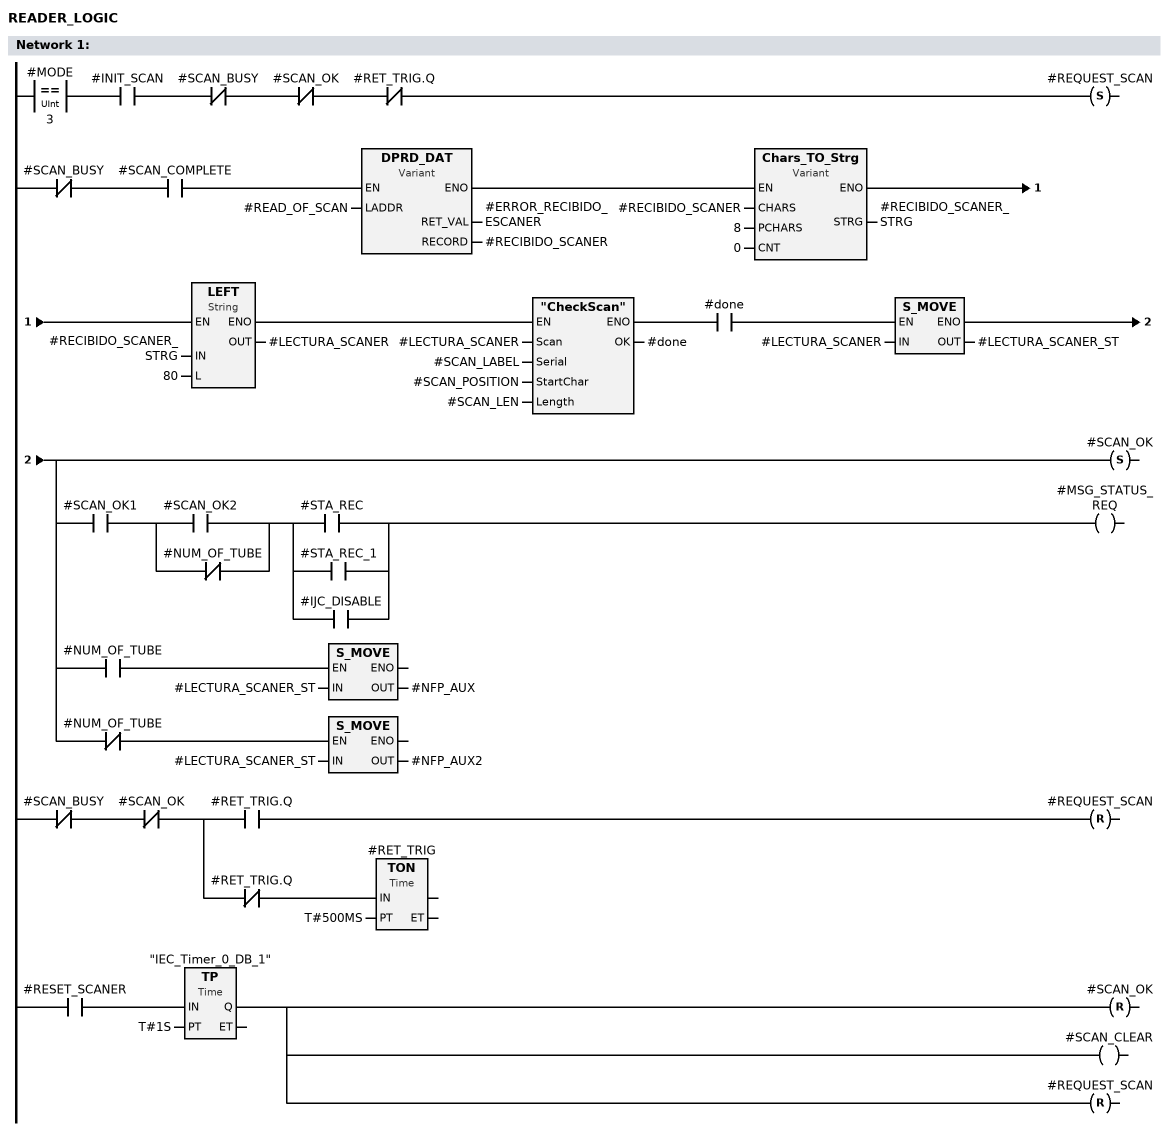
   RUNG wire#powerrail
      { S7_Templates := "SrcType := UInt" } EQ_Contact(in1 := #MODE, in2 := 3)
      Contact( #INIT_SCAN )
      I_Contact( #SCAN_BUSY )
      I_Contact( #SCAN_OK )
      I_Contact( #RET_TRIG.Q )
      S_Coil( #REQUEST_SCAN )
   END_RUNG
   RUNG wire#powerrail
      I_Contact( #SCAN_BUSY )
      Contact( #SCAN_COMPLETE )
      { S7_Templates := "[ptr_type := Variant, laddr_type := HW_IO]" } DPRD_DAT(LADDR := #READ_OF_SCAN, RET_VAL => #ERROR_RECIBIDO_ESCANER, RECORD => #RECIBIDO_SCANER)
      { S7_Templates := "[ptr_type := Variant, str_type := String]" } Chars_TO_Strg(Chars := #RECIBIDO_SCANER, pChars := 8, Cnt := 0, Strg => #RECIBIDO_SCANER_STRG)
      { S7_Templates := "str_type := String" } LEFT(IN := #RECIBIDO_SCANER_STRG, L := 80, OUT => #LECTURA_SCANER)
      "CheckScan"(Scan := #LECTURA_SCANER, Serial := #SCAN_LABEL, StartChar := #SCAN_POSITION, Length := #SCAN_LEN, OK => #done)
      Contact( #done )
      S_Move(in := #LECTURA_SCANER, out => #LECTURA_SCANER_ST)
      wire#w1
      S_Coil( #SCAN_OK )
   END_RUNG
   RUNG wire#w1
      Contact( #SCAN_OK1 )
      wire#w2
      Contact( #SCAN_OK2 )
      wire#w3
      Contact( #STA_REC )
      wire#w4
      Coil( #MSG_STATUS_REQ )
   END_RUNG
   RUNG wire#w2
      I_Contact( #NUM_OF_TUBE )
   END_RUNG wire#w3
   RUNG wire#w3
      Contact( #STA_REC_1 )
   END_RUNG wire#w4
   RUNG wire#w3
      Contact( #IJC_DISABLE )
   END_RUNG wire#w4
   RUNG wire#w1
      Contact( #NUM_OF_TUBE )
      S_Move(in := #LECTURA_SCANER_ST, out => #NFP_AUX)
   END_RUNG
   RUNG wire#w1
      I_Contact( #NUM_OF_TUBE )
      S_Move(in := #LECTURA_SCANER_ST, out => #NFP_AUX2)
   END_RUNG
   RUNG wire#powerrail
      I_Contact( #SCAN_BUSY )
      I_Contact( #SCAN_OK )
      wire#w5
      Contact( #RET_TRIG.Q )
      R_Coil( #REQUEST_SCAN )
   END_RUNG
   RUNG wire#w5
      I_Contact( #RET_TRIG.Q )
      { S7_Templates := "time_type := Time" } #RET_TRIG.TON(pt := T#500MS, et =>)
   END_RUNG
   RUNG wire#powerrail
      Contact( #RESET_SCANER )
      { S7_Templates := "time_type := Time" } "IEC_Timer_0_DB_1".TP(pt := T#1S, et =>)
      wire#w6
      R_Coil( #SCAN_OK )
   END_RUNG
   RUNG wire#w6
      Coil( #SCAN_CLEAR )
   END_RUNG
   RUNG wire#w6
      R_Coil( #REQUEST_SCAN )
   END_RUNG
   // the same network as SCL:
   IF (#MODE = 3) AND #INIT_SCAN AND NOT #SCAN_BUSY AND NOT #SCAN_OK AND NOT #RET_TRIG.Q THEN
       #REQUEST_SCAN := TRUE;
   END_IF;
   #ERROR_RECIBIDO_ESCANER := DPRD_DAT(EN := NOT #SCAN_BUSY AND #SCAN_COMPLETE,
                           LADDR := #READ_OF_SCAN,
                           RECORD => #RECIBIDO_SCANER,
                           ENO => #_w1);
   Chars_TO_Strg(EN := #_w1,
                 Chars := #RECIBIDO_SCANER,
                 pChars := 8,
                 Cnt := 0,
                 Strg => #RECIBIDO_SCANER_STRG,
                 ENO => #_w2);
   LEFT(EN := #_w2, IN := #RECIBIDO_SCANER_STRG, L := 80, OUT => #LECTURA_SCANER, ENO => #_w3);
   "CheckScan"(EN := #_w3,
               Scan := #LECTURA_SCANER,
               Serial := #SCAN_LABEL,
               StartChar := #SCAN_POSITION,
               Length := #SCAN_LEN,
               OK => #done,
               ENO => #_w4);
   #_w5 := #_w4 AND #done;
   IF #_w5 THEN
       #LECTURA_SCANER_ST := #LECTURA_SCANER;
       #SCAN_OK := TRUE;
   END_IF;
   #MSG_STATUS_REQ := #_w5 AND #SCAN_OK1 AND (#SCAN_OK2 OR NOT #NUM_OF_TUBE) AND (#STA_REC OR #STA_REC_1 OR #IJC_DISABLE);
   IF #_w5 AND #NUM_OF_TUBE THEN #NFP_AUX := #LECTURA_SCANER_ST; END_IF;
   IF #_w5 AND NOT #NUM_OF_TUBE THEN #NFP_AUX2 := #LECTURA_SCANER_ST; END_IF;
   #_w6 := NOT #SCAN_BUSY AND NOT #SCAN_OK;
   IF #_w6 AND #RET_TRIG.Q THEN #REQUEST_SCAN := FALSE; END_IF;
   #RET_TRIG.TON(IN := #_w6 AND NOT #RET_TRIG.Q, PT := T#500MS);
   "IEC_Timer_0_DB_1".TP(IN := #RESET_SCANER, PT := T#1S);
   IF "IEC_Timer_0_DB_1".Q THEN #SCAN_OK := FALSE; END_IF;
   #SCAN_CLEAR := "IEC_Timer_0_DB_1".Q;
   IF "IEC_Timer_0_DB_1".Q THEN #REQUEST_SCAN := FALSE; END_IF;
END_REGION
END_FUNCTION_BLOCK

FUNCTION "CylinderCollisions" : Void
{ S7_Optimized_Access := 'TRUE' }
VERSION : 0.1

BEGIN
	
	//***************** Collisions calls *****************
	
	REGION "CylinderGeneratedCalls_DB".MM2200_GrippingTubeFrontInstant
	    // Call Cylinder control "CylinderGeneratedCalls_DB".MM2200_GrippingTubeFrontInstantr
	    "CylinderGeneratedCalls_DB".MM2200_GrippingTubeFrontInstant.iNoCollisionBasic := true;
	    "CylinderGeneratedCalls_DB".MM2200_GrippingTubeFrontInstant.iNoCollisionWork := true;
	    "CylinderGeneratedCalls_DB".MM2200_GrippingTubeFrontInstant.iNoCollisionFree := true;
	END_REGION
	
	REGION "CylinderGeneratedCalls_DB".MM2201_GrippingTubeRearInstant
	    // Call Cylinder control "CylinderGeneratedCalls_DB".MM2201_GrippingTubeRearInstantr
	    "CylinderGeneratedCalls_DB".MM2201_GrippingTubeRearInstant.iNoCollisionBasic := true;
	    "CylinderGeneratedCalls_DB".MM2201_GrippingTubeRearInstant.iNoCollisionWork := true;
	    "CylinderGeneratedCalls_DB".MM2201_GrippingTubeRearInstant.iNoCollisionFree := true;
	END_REGION
	
	REGION "CylinderGeneratedCalls_DB".MM2220_HoldingSidememberInsideLeftInstant
	    // Call Cylinder control "CylinderGeneratedCalls_DB".MM2220_HoldingSidememberInsideLeftInstantr
	    "CylinderGeneratedCalls_DB".MM2220_HoldingSidememberInsideLeftInstant.iNoCollisionBasic := true;
	    "CylinderGeneratedCalls_DB".MM2220_HoldingSidememberInsideLeftInstant.iNoCollisionWork := true;
	    "CylinderGeneratedCalls_DB".MM2220_HoldingSidememberInsideLeftInstant.iNoCollisionFree := true;
	END_REGION
	
	REGION "CylinderGeneratedCalls_DB".MM2221_HoldingSidememberInsideRightInstant
	    // Call Cylinder control "CylinderGeneratedCalls_DB".MM2221_HoldingSidememberInsideRightInstantr
	    "CylinderGeneratedCalls_DB".MM2221_HoldingSidememberInsideRightInstant.iNoCollisionBasic := true;
	    "CylinderGeneratedCalls_DB".MM2221_HoldingSidememberInsideRightInstant.iNoCollisionWork := true;
	    "CylinderGeneratedCalls_DB".MM2221_HoldingSidememberInsideRightInstant.iNoCollisionFree := true;
	END_REGION
	
	REGION "CylinderGeneratedCalls_DB".MM2240_HoldingSidememberOutsideLeftInstant
	    // Call Cylinder control "CylinderGeneratedCalls_DB".MM2240_HoldingSidememberOutsideLeftInstantr
	    "CylinderGeneratedCalls_DB".MM2240_HoldingSidememberOutsideLeftInstant.iNoCollisionBasic := true;
	    "CylinderGeneratedCalls_DB".MM2240_HoldingSidememberOutsideLeftInstant.iNoCollisionWork := true;
	    "CylinderGeneratedCalls_DB".MM2240_HoldingSidememberOutsideLeftInstant.iNoCollisionFree := true;
	END_REGION
	
	REGION "CylinderGeneratedCalls_DB".MM2241_HoldingSidememberOutsideRightInstant
	    // Call Cylinder control "CylinderGeneratedCalls_DB".MM2241_HoldingSidememberOutsideRightInstantr
	    "CylinderGeneratedCalls_DB".MM2241_HoldingSidememberOutsideRightInstant.iNoCollisionBasic := true;
	    "CylinderGeneratedCalls_DB".MM2241_HoldingSidememberOutsideRightInstant.iNoCollisionWork := true;
	    "CylinderGeneratedCalls_DB".MM2241_HoldingSidememberOutsideRightInstant.iNoCollisionFree := true;
	END_REGION
	
	REGION "CylinderGeneratedCalls_DB".MM2500_GrippingTubeFrontInstant
	    // Call Cylinder control "CylinderGeneratedCalls_DB".MM2500_GrippingTubeFrontInstantr
	    "CylinderGeneratedCalls_DB".MM2500_GrippingTubeFrontInstant.iNoCollisionBasic := true;
	    "CylinderGeneratedCalls_DB".MM2500_GrippingTubeFrontInstant.iNoCollisionWork := true;
	    "CylinderGeneratedCalls_DB".MM2500_GrippingTubeFrontInstant.iNoCollisionFree := true;
	END_REGION
	
	REGION "CylinderGeneratedCalls_DB".MM2501_GrippingTubeRearInstant
	    // Call Cylinder control "CylinderGeneratedCalls_DB".MM2501_GrippingTubeRearInstantr
	    "CylinderGeneratedCalls_DB".MM2501_GrippingTubeRearInstant.iNoCollisionBasic := true;
	    "CylinderGeneratedCalls_DB".MM2501_GrippingTubeRearInstant.iNoCollisionWork := true;
	    "CylinderGeneratedCalls_DB".MM2501_GrippingTubeRearInstant.iNoCollisionFree := true;
	END_REGION
	
	REGION "CylinderGeneratedCalls_DB".MM2520_HoldingSidememberInsideLeftInstant
	    // Call Cylinder control "CylinderGeneratedCalls_DB".MM2520_HoldingSidememberInsideLeftInstantr
	    "CylinderGeneratedCalls_DB".MM2520_HoldingSidememberInsideLeftInstant.iNoCollisionBasic := true;
	    "CylinderGeneratedCalls_DB".MM2520_HoldingSidememberInsideLeftInstant.iNoCollisionWork := true;
	    "CylinderGeneratedCalls_DB".MM2520_HoldingSidememberInsideLeftInstant.iNoCollisionFree := true;
	END_REGION
	
	REGION "CylinderGeneratedCalls_DB".MM2521_HoldingSidememberInsideRightInstant
	    // Call Cylinder control "CylinderGeneratedCalls_DB".MM2521_HoldingSidememberInsideRightInstantr
	    "CylinderGeneratedCalls_DB".MM2521_HoldingSidememberInsideRightInstant.iNoCollisionBasic := true;
	    "CylinderGeneratedCalls_DB".MM2521_HoldingSidememberInsideRightInstant.iNoCollisionWork := true;
	    "CylinderGeneratedCalls_DB".MM2521_HoldingSidememberInsideRightInstant.iNoCollisionFree := true;
	END_REGION
	
	REGION "CylinderGeneratedCalls_DB".MM2540_HoldingSidememberOutsideLeftInstant
	    // Call Cylinder control "CylinderGeneratedCalls_DB".MM2540_HoldingSidememberOutsideLeftInstantr
	    "CylinderGeneratedCalls_DB".MM2540_HoldingSidememberOutsideLeftInstant.iNoCollisionBasic := true;
	    "CylinderGeneratedCalls_DB".MM2540_HoldingSidememberOutsideLeftInstant.iNoCollisionWork := true;
	    "CylinderGeneratedCalls_DB".MM2540_HoldingSidememberOutsideLeftInstant.iNoCollisionFree := true;
	END_REGION
	
	REGION "CylinderGeneratedCalls_DB".MM2541_HoldingSidememberOutsideRightInstant
	    // Call Cylinder control "CylinderGeneratedCalls_DB".MM2541_HoldingSidememberOutsideRightInstantr
	    "CylinderGeneratedCalls_DB".MM2541_HoldingSidememberOutsideRightInstant.iNoCollisionBasic := true;
	    "CylinderGeneratedCalls_DB".MM2541_HoldingSidememberOutsideRightInstant.iNoCollisionWork := true;
	    "CylinderGeneratedCalls_DB".MM2541_HoldingSidememberOutsideRightInstant.iNoCollisionFree := true;
	END_REGION
	
	REGION "CylinderGeneratedCalls_DB".MM300_ShiftingSupportRightInstant
	    // Call Cylinder control "CylinderGeneratedCalls_DB".MM300_ShiftingSupportRightInstantr
	    "CylinderGeneratedCalls_DB".MM300_ShiftingSupportRightInstant.iNoCollisionBasic := true;
	    "CylinderGeneratedCalls_DB".MM300_ShiftingSupportRightInstant.iNoCollisionWork := true;
	    "CylinderGeneratedCalls_DB".MM300_ShiftingSupportRightInstant.iNoCollisionFree := true;
	END_REGION
	
	REGION "CylinderGeneratedCalls_DB".MM302_ShiftingSupportLeftInstant
	    // Call Cylinder control "CylinderGeneratedCalls_DB".MM302_ShiftingSupportLeftInstantr
	    "CylinderGeneratedCalls_DB".MM302_ShiftingSupportLeftInstant.iNoCollisionBasic := true;
	    "CylinderGeneratedCalls_DB".MM302_ShiftingSupportLeftInstant.iNoCollisionWork := true;
	    "CylinderGeneratedCalls_DB".MM302_ShiftingSupportLeftInstant.iNoCollisionFree := true;
	END_REGION
	
	REGION "CylinderGeneratedCalls_DB".MM304_MovingStopRightInstant
	    // Call Cylinder control "CylinderGeneratedCalls_DB".MM304_MovingStopRightInstantr
	    "CylinderGeneratedCalls_DB".MM304_MovingStopRightInstant.iNoCollisionBasic := "DevicesData".Cylinders["MM304_MovingStopRight"].InBp OR
	    "DevicesData".Cylinders["MM350_ShiftWedgeRight"].InBp;
	    "CylinderGeneratedCalls_DB".MM304_MovingStopRightInstant.iNoCollisionWork := "DevicesData".Cylinders["MM304_MovingStopRight"].InWp OR
	    "DevicesData".Cylinders["MM350_ShiftWedgeRight"].InBp;;
	    "CylinderGeneratedCalls_DB".MM304_MovingStopRightInstant.iNoCollisionFree := true;
	END_REGION
	
	REGION "CylinderGeneratedCalls_DB".MM306_MovingStopLeftInstant
	    // Call Cylinder control "CylinderGeneratedCalls_DB".MM306_MovingStopLeftInstantr
	    "CylinderGeneratedCalls_DB".MM306_MovingStopLeftInstant.iNoCollisionBasic := "DevicesData".Cylinders["MM306_MovingStopLeft"].InBp OR
	    "DevicesData".Cylinders["MM352_ShiftWedgeLeft"].InBp;
	    "CylinderGeneratedCalls_DB".MM306_MovingStopLeftInstant.iNoCollisionWork := "DevicesData".Cylinders["MM306_MovingStopLeft"].InWp OR
	    "DevicesData".Cylinders["MM352_ShiftWedgeLeft"].InBp;
	    "CylinderGeneratedCalls_DB".MM306_MovingStopLeftInstant.iNoCollisionFree := true;
	END_REGION
	
	REGION "CylinderGeneratedCalls_DB".MM340_RivetingUnitRightInstant
	    // Call Cylinder control "CylinderGeneratedCalls_DB".MM340_RivetingUnitRightInstantr
	    "CylinderGeneratedCalls_DB".MM340_RivetingUnitRightInstant.iNoCollisionBasic := "DevicesData".Cylinders["MM344_RivetingSupportRight"].InBp;
	    "CylinderGeneratedCalls_DB".MM340_RivetingUnitRightInstant.iNoCollisionWork := "DevicesData".Cylinders["MM344_RivetingSupportRight"].InBp;
	    "CylinderGeneratedCalls_DB".MM340_RivetingUnitRightInstant.iNoCollisionFree := true;
	END_REGION
	
	REGION "CylinderGeneratedCalls_DB".MM342_RivetingUnitLeftInstant
	    // Call Cylinder control "CylinderGeneratedCalls_DB".MM342_RivetingUnitLeftInstantr
	    "CylinderGeneratedCalls_DB".MM342_RivetingUnitLeftInstant.iNoCollisionBasic := "DevicesData".Cylinders["MM346_RivetingSupportLeft"].InBp;
	    "CylinderGeneratedCalls_DB".MM342_RivetingUnitLeftInstant.iNoCollisionWork := "DevicesData".Cylinders["MM346_RivetingSupportLeft"].InBp;
	    "CylinderGeneratedCalls_DB".MM342_RivetingUnitLeftInstant.iNoCollisionFree := true;
	END_REGION
	
	REGION "CylinderGeneratedCalls_DB".MM344_RivetingSupportRightInstant
	    // Call Cylinder control "CylinderGeneratedCalls_DB".MM344_RivetingSupportRightInstantr
	    "CylinderGeneratedCalls_DB".MM344_RivetingSupportRightInstant.iNoCollisionBasic := true;
	    "CylinderGeneratedCalls_DB".MM344_RivetingSupportRightInstant.iNoCollisionWork := true;
	    "CylinderGeneratedCalls_DB".MM344_RivetingSupportRightInstant.iNoCollisionFree := true;
	END_REGION
	
	REGION "CylinderGeneratedCalls_DB".MM346_RivetingSupportLeftInstant
	    // Call Cylinder control "CylinderGeneratedCalls_DB".MM346_RivetingSupportLeftInstantr
	    "CylinderGeneratedCalls_DB".MM346_RivetingSupportLeftInstant.iNoCollisionBasic := true;
	    "CylinderGeneratedCalls_DB".MM346_RivetingSupportLeftInstant.iNoCollisionWork := true;
	    "CylinderGeneratedCalls_DB".MM346_RivetingSupportLeftInstant.iNoCollisionFree := true;
	END_REGION
	
	REGION "CylinderGeneratedCalls_DB".MM350_ShiftWedgeRightInstant
	    // Call Cylinder control "CylinderGeneratedCalls_DB".MM350_ShiftWedgeRightInstantr
	    "CylinderGeneratedCalls_DB".MM350_ShiftWedgeRightInstant.iNoCollisionBasic := true;
	    "CylinderGeneratedCalls_DB".MM350_ShiftWedgeRightInstant.iNoCollisionWork := true;
	    "CylinderGeneratedCalls_DB".MM350_ShiftWedgeRightInstant.iNoCollisionFree := true;
	END_REGION
	
	REGION "CylinderGeneratedCalls_DB".MM352_ShiftWedgeLeftInstant
	    // Call Cylinder control "CylinderGeneratedCalls_DB".MM352_ShiftWedgeLeftInstantr
	    "CylinderGeneratedCalls_DB".MM352_ShiftWedgeLeftInstant.iNoCollisionBasic := true;
	    "CylinderGeneratedCalls_DB".MM352_ShiftWedgeLeftInstant.iNoCollisionWork := true;
	    "CylinderGeneratedCalls_DB".MM352_ShiftWedgeLeftInstant.iNoCollisionFree := true;
	END_REGION
	
	REGION "CylinderGeneratedCalls_DB".MM104_AutoejectGripperLiftingInstant
	    // Call Cylinder control "CylinderGeneratedCalls_DB".MM104_AutoejectGripperLiftingInstantr
	    "CylinderGeneratedCalls_DB".MM104_AutoejectGripperLiftingInstant.iNoCollisionBasic := true;
	    "CylinderGeneratedCalls_DB".MM104_AutoejectGripperLiftingInstant.iNoCollisionWork :=
	    "DevicesData"."TA1-3MA".data.zones.inNOKpos
	    OR
	    "DevicesData"."TA1-3MA".data.zones.inOKpos AND
	    (NOT "i4partPresent" OR
	    "DevicesData".Cylinders["MM2500_GrippingTubeFront"].InBp AND
	    "DevicesData".Cylinders["MM2520_HoldingSidememberInsideLeft"].InBp AND
	    "DevicesData".Cylinders["MM2540_HoldingSidememberOutsideLeft"].InBp)
	    OR
	    "DevicesData"."TA1-3MA".data.zones.inST3jig AND
	    (NOT "i3partPresent" OR
	    "DevicesData".Cylinders["MM2500_GrippingTubeFront"].InBp AND
	    "DevicesData".Cylinders["MM2520_HoldingSidememberInsideLeft"].InBp AND
	    "DevicesData".Cylinders["MM2540_HoldingSidememberOutsideLeft"].InBp) AND
	    "DevicesData".Cylinders["MM300_ShiftingSupportRight"].InBp AND
	    "DevicesData".Cylinders["MM302_ShiftingSupportLeft"].InBp AND
	    "DevicesData".Cylinders["MM340_RivetingUnitRight"].InBp AND
	    "DevicesData".Cylinders["MM342_RivetingUnitLeft"].InBp AND
	    "DevicesData".Cylinders["MM344_RivetingSupportRight"].InBp AND
	    "DevicesData".Cylinders["MM346_RivetingSupportLeft"].InBp;
	    "CylinderGeneratedCalls_DB".MM104_AutoejectGripperLiftingInstant.iNoCollisionFree := true;
	END_REGION
	
	REGION "CylinderGeneratedCalls_DB".MM3100_SidememberSupportLeftInstant
	    // Call Cylinder control "CylinderGeneratedCalls_DB".MM3100_SidememberSupportLeftInstantr
	    "CylinderGeneratedCalls_DB".MM3100_SidememberSupportLeftInstant.iNoCollisionBasic := true;
	    "CylinderGeneratedCalls_DB".MM3100_SidememberSupportLeftInstant.iNoCollisionWork := true;
	    "CylinderGeneratedCalls_DB".MM3100_SidememberSupportLeftInstant.iNoCollisionFree := true;
	END_REGION
	
	REGION "CylinderGeneratedCalls_DB".MM3101_SidememberSupportRightInstant
	    // Call Cylinder control "CylinderGeneratedCalls_DB".MM3101_SidememberSupportRightInstantr
	    "CylinderGeneratedCalls_DB".MM3101_SidememberSupportRightInstant.iNoCollisionBasic := true;
	    "CylinderGeneratedCalls_DB".MM3101_SidememberSupportRightInstant.iNoCollisionWork := true;
	    "CylinderGeneratedCalls_DB".MM3101_SidememberSupportRightInstant.iNoCollisionFree := true;
	END_REGION
	
	//***************** timing and safety calls *****************
	
	REGION "CylinderGeneratedCalls_DB".MM2200_GrippingTubeFrontInstant
	    // Call Cylinder control "CylinderGeneratedCalls_DB".MM2200_GrippingTubeFrontInstantr
	    "CylinderGeneratedCalls_DB".MM2200_GrippingTubeFrontInstant.POWER_OK := "safety_signals"."3L+" OR TRUE;
	    "CylinderGeneratedCalls_DB".MM2200_GrippingTubeFrontInstant.DELAY_BASIC := t#100ms;
	    "CylinderGeneratedCalls_DB".MM2200_GrippingTubeFrontInstant.DELAY_WORK := t#100ms;
	    "CylinderGeneratedCalls_DB".MM2200_GrippingTubeFrontInstant.DELAY_FREE := T#100mS;
	    "CylinderGeneratedCalls_DB".MM2200_GrippingTubeFrontInstant.ERROR_TIME := T#10S;
	    "CylinderGeneratedCalls_DB".MM2200_GrippingTubeFrontInstant.ValveDelay := T#0ms;
	END_REGION
	
	REGION "CylinderGeneratedCalls_DB".MM2201_GrippingTubeRearInstant
	    // Call Cylinder control "CylinderGeneratedCalls_DB".MM2201_GrippingTubeRearInstantr
	    "CylinderGeneratedCalls_DB".MM2201_GrippingTubeRearInstant.POWER_OK := "safety_signals"."3L+" OR TRUE;
	    "CylinderGeneratedCalls_DB".MM2201_GrippingTubeRearInstant.DELAY_BASIC := t#100ms;
	    "CylinderGeneratedCalls_DB".MM2201_GrippingTubeRearInstant.DELAY_WORK := t#100ms;
	    "CylinderGeneratedCalls_DB".MM2201_GrippingTubeRearInstant.DELAY_FREE := T#100mS;
	    "CylinderGeneratedCalls_DB".MM2201_GrippingTubeRearInstant.ERROR_TIME := T#10S;
	    "CylinderGeneratedCalls_DB".MM2201_GrippingTubeRearInstant.ValveDelay := T#0ms;
	END_REGION
	
	REGION "CylinderGeneratedCalls_DB".MM2220_HoldingSidememberInsideLeftInstant
	    // Call Cylinder control "CylinderGeneratedCalls_DB".MM2220_HoldingSidememberInsideLeftInstantr
	    "CylinderGeneratedCalls_DB".MM2220_HoldingSidememberInsideLeftInstant.POWER_OK := "safety_signals"."3L+" OR TRUE;
	    "CylinderGeneratedCalls_DB".MM2220_HoldingSidememberInsideLeftInstant.DELAY_BASIC := t#100ms;
	    "CylinderGeneratedCalls_DB".MM2220_HoldingSidememberInsideLeftInstant.DELAY_WORK := t#100ms;
	    "CylinderGeneratedCalls_DB".MM2220_HoldingSidememberInsideLeftInstant.DELAY_FREE := T#100mS;
	    "CylinderGeneratedCalls_DB".MM2220_HoldingSidememberInsideLeftInstant.ERROR_TIME := T#10S;
	    "CylinderGeneratedCalls_DB".MM2220_HoldingSidememberInsideLeftInstant.ValveDelay := T#0ms;
	END_REGION
	
	REGION "CylinderGeneratedCalls_DB".MM2221_HoldingSidememberInsideRightInstant
	    // Call Cylinder control "CylinderGeneratedCalls_DB".MM2221_HoldingSidememberInsideRightInstantr
	    "CylinderGeneratedCalls_DB".MM2221_HoldingSidememberInsideRightInstant.POWER_OK := "safety_signals"."3L+" OR TRUE;
	    "CylinderGeneratedCalls_DB".MM2221_HoldingSidememberInsideRightInstant.DELAY_BASIC := t#100ms;
	    "CylinderGeneratedCalls_DB".MM2221_HoldingSidememberInsideRightInstant.DELAY_WORK := t#100ms;
	    "CylinderGeneratedCalls_DB".MM2221_HoldingSidememberInsideRightInstant.DELAY_FREE := T#100mS;
	    "CylinderGeneratedCalls_DB".MM2221_HoldingSidememberInsideRightInstant.ERROR_TIME := T#10S;
	    "CylinderGeneratedCalls_DB".MM2221_HoldingSidememberInsideRightInstant.ValveDelay := T#0ms;
	END_REGION
	
	REGION "CylinderGeneratedCalls_DB".MM2240_HoldingSidememberOutsideLeftInstant
	    // Call Cylinder control "CylinderGeneratedCalls_DB".MM2240_HoldingSidememberOutsideLeftInstantr
	    "CylinderGeneratedCalls_DB".MM2240_HoldingSidememberOutsideLeftInstant.POWER_OK := "safety_signals"."3L+" OR TRUE;
	    "CylinderGeneratedCalls_DB".MM2240_HoldingSidememberOutsideLeftInstant.DELAY_BASIC := t#100ms;
	    "CylinderGeneratedCalls_DB".MM2240_HoldingSidememberOutsideLeftInstant.DELAY_WORK := t#100ms;
	    "CylinderGeneratedCalls_DB".MM2240_HoldingSidememberOutsideLeftInstant.DELAY_FREE := T#100mS;
	    "CylinderGeneratedCalls_DB".MM2240_HoldingSidememberOutsideLeftInstant.ERROR_TIME := T#10S;
	    "CylinderGeneratedCalls_DB".MM2240_HoldingSidememberOutsideLeftInstant.ValveDelay := T#0ms;
	END_REGION
	
	REGION "CylinderGeneratedCalls_DB".MM2241_HoldingSidememberOutsideRightInstant
	    // Call Cylinder control "CylinderGeneratedCalls_DB".MM2241_HoldingSidememberOutsideRightInstantr
	    "CylinderGeneratedCalls_DB".MM2241_HoldingSidememberOutsideRightInstant.POWER_OK := "safety_signals"."3L+" OR TRUE;
	    "CylinderGeneratedCalls_DB".MM2241_HoldingSidememberOutsideRightInstant.DELAY_BASIC := t#100ms;
	    "CylinderGeneratedCalls_DB".MM2241_HoldingSidememberOutsideRightInstant.DELAY_WORK := t#100ms;
	    "CylinderGeneratedCalls_DB".MM2241_HoldingSidememberOutsideRightInstant.DELAY_FREE := T#100mS;
	    "CylinderGeneratedCalls_DB".MM2241_HoldingSidememberOutsideRightInstant.ERROR_TIME := T#10S;
	    "CylinderGeneratedCalls_DB".MM2241_HoldingSidememberOutsideRightInstant.ValveDelay := T#0ms;
	END_REGION
	
	REGION "CylinderGeneratedCalls_DB".MM2500_GrippingTubeFrontInstant
	    // Call Cylinder control "CylinderGeneratedCalls_DB".MM2500_GrippingTubeFrontInstantr
	    "CylinderGeneratedCalls_DB".MM2500_GrippingTubeFrontInstant.POWER_OK := true;
	    "CylinderGeneratedCalls_DB".MM2500_GrippingTubeFrontInstant.DELAY_BASIC := t#100ms;
	    "CylinderGeneratedCalls_DB".MM2500_GrippingTubeFrontInstant.DELAY_WORK := t#100ms;
	    "CylinderGeneratedCalls_DB".MM2500_GrippingTubeFrontInstant.DELAY_FREE := T#100mS;
	    "CylinderGeneratedCalls_DB".MM2500_GrippingTubeFrontInstant.ERROR_TIME := T#10S;
	    "CylinderGeneratedCalls_DB".MM2500_GrippingTubeFrontInstant.ValveDelay := T#0ms;
	END_REGION
	
	REGION "CylinderGeneratedCalls_DB".MM2501_GrippingTubeRearInstant
	    // Call Cylinder control "CylinderGeneratedCalls_DB".MM2501_GrippingTubeRearInstantr
	    "CylinderGeneratedCalls_DB".MM2501_GrippingTubeRearInstant.POWER_OK := true;
	    "CylinderGeneratedCalls_DB".MM2501_GrippingTubeRearInstant.DELAY_BASIC := t#100ms;
	    "CylinderGeneratedCalls_DB".MM2501_GrippingTubeRearInstant.DELAY_WORK := t#100ms;
	    "CylinderGeneratedCalls_DB".MM2501_GrippingTubeRearInstant.DELAY_FREE := T#100mS;
	    "CylinderGeneratedCalls_DB".MM2501_GrippingTubeRearInstant.ERROR_TIME := T#10S;
	    "CylinderGeneratedCalls_DB".MM2501_GrippingTubeRearInstant.ValveDelay := T#0ms;
	END_REGION
	
	REGION "CylinderGeneratedCalls_DB".MM2520_HoldingSidememberInsideLeftInstant
	    // Call Cylinder control "CylinderGeneratedCalls_DB".MM2520_HoldingSidememberInsideLeftInstantr
	    "CylinderGeneratedCalls_DB".MM2520_HoldingSidememberInsideLeftInstant.POWER_OK := true;
	    "CylinderGeneratedCalls_DB".MM2520_HoldingSidememberInsideLeftInstant.DELAY_BASIC := t#100ms;
	    "CylinderGeneratedCalls_DB".MM2520_HoldingSidememberInsideLeftInstant.DELAY_WORK := t#100ms;
	    "CylinderGeneratedCalls_DB".MM2520_HoldingSidememberInsideLeftInstant.DELAY_FREE := T#100mS;
	    "CylinderGeneratedCalls_DB".MM2520_HoldingSidememberInsideLeftInstant.ERROR_TIME := T#10S;
	    "CylinderGeneratedCalls_DB".MM2520_HoldingSidememberInsideLeftInstant.ValveDelay := T#0ms;
	END_REGION
	
	REGION "CylinderGeneratedCalls_DB".MM2521_HoldingSidememberInsideRightInstant
	    // Call Cylinder control "CylinderGeneratedCalls_DB".MM2521_HoldingSidememberInsideRightInstantr
	    "CylinderGeneratedCalls_DB".MM2521_HoldingSidememberInsideRightInstant.POWER_OK := true;
	    "CylinderGeneratedCalls_DB".MM2521_HoldingSidememberInsideRightInstant.DELAY_BASIC := t#100ms;
	    "CylinderGeneratedCalls_DB".MM2521_HoldingSidememberInsideRightInstant.DELAY_WORK := t#100ms;
	    "CylinderGeneratedCalls_DB".MM2521_HoldingSidememberInsideRightInstant.DELAY_FREE := T#100mS;
	    "CylinderGeneratedCalls_DB".MM2521_HoldingSidememberInsideRightInstant.ERROR_TIME := T#10S;
	    "CylinderGeneratedCalls_DB".MM2521_HoldingSidememberInsideRightInstant.ValveDelay := T#0ms;
	END_REGION
	
	REGION "CylinderGeneratedCalls_DB".MM2540_HoldingSidememberOutsideLeftInstant
	    // Call Cylinder control "CylinderGeneratedCalls_DB".MM2540_HoldingSidememberOutsideLeftInstantr
	    "CylinderGeneratedCalls_DB".MM2540_HoldingSidememberOutsideLeftInstant.POWER_OK := true;
	    "CylinderGeneratedCalls_DB".MM2540_HoldingSidememberOutsideLeftInstant.DELAY_BASIC := t#100ms;
	    "CylinderGeneratedCalls_DB".MM2540_HoldingSidememberOutsideLeftInstant.DELAY_WORK := t#100ms;
	    "CylinderGeneratedCalls_DB".MM2540_HoldingSidememberOutsideLeftInstant.DELAY_FREE := T#100mS;
	    "CylinderGeneratedCalls_DB".MM2540_HoldingSidememberOutsideLeftInstant.ERROR_TIME := T#10S;
	    "CylinderGeneratedCalls_DB".MM2540_HoldingSidememberOutsideLeftInstant.ValveDelay := T#0ms;
	END_REGION
	
	REGION "CylinderGeneratedCalls_DB".MM2541_HoldingSidememberOutsideRightInstant
	    // Call Cylinder control "CylinderGeneratedCalls_DB".MM2541_HoldingSidememberOutsideRightInstantr
	    "CylinderGeneratedCalls_DB".MM2541_HoldingSidememberOutsideRightInstant.POWER_OK := true;
	    "CylinderGeneratedCalls_DB".MM2541_HoldingSidememberOutsideRightInstant.DELAY_BASIC := t#100ms;
	    "CylinderGeneratedCalls_DB".MM2541_HoldingSidememberOutsideRightInstant.DELAY_WORK := t#100ms;
	    "CylinderGeneratedCalls_DB".MM2541_HoldingSidememberOutsideRightInstant.DELAY_FREE := T#100mS;
	    "CylinderGeneratedCalls_DB".MM2541_HoldingSidememberOutsideRightInstant.ERROR_TIME := T#10S;
	    "CylinderGeneratedCalls_DB".MM2541_HoldingSidememberOutsideRightInstant.ValveDelay := T#0ms;
	END_REGION
	
	REGION "CylinderGeneratedCalls_DB".MM300_ShiftingSupportRightInstant
	    // Call Cylinder control "CylinderGeneratedCalls_DB".MM300_ShiftingSupportRightInstantr
	    "CylinderGeneratedCalls_DB".MM300_ShiftingSupportRightInstant.POWER_OK := true;
	    "CylinderGeneratedCalls_DB".MM300_ShiftingSupportRightInstant.DELAY_BASIC := t#100ms;
	    "CylinderGeneratedCalls_DB".MM300_ShiftingSupportRightInstant.DELAY_WORK := t#100ms;
	    "CylinderGeneratedCalls_DB".MM300_ShiftingSupportRightInstant.DELAY_FREE := T#100mS;
	    "CylinderGeneratedCalls_DB".MM300_ShiftingSupportRightInstant.ERROR_TIME := T#10S;
	    "CylinderGeneratedCalls_DB".MM300_ShiftingSupportRightInstant.ValveDelay := T#0ms;
	END_REGION
	
	REGION "CylinderGeneratedCalls_DB".MM302_ShiftingSupportLeftInstant
	    // Call Cylinder control "CylinderGeneratedCalls_DB".MM302_ShiftingSupportLeftInstantr
	    "CylinderGeneratedCalls_DB".MM302_ShiftingSupportLeftInstant.POWER_OK := true;
	    "CylinderGeneratedCalls_DB".MM302_ShiftingSupportLeftInstant.DELAY_BASIC := t#100ms;
	    "CylinderGeneratedCalls_DB".MM302_ShiftingSupportLeftInstant.DELAY_WORK := t#100ms;
	    "CylinderGeneratedCalls_DB".MM302_ShiftingSupportLeftInstant.DELAY_FREE := T#100mS;
	    "CylinderGeneratedCalls_DB".MM302_ShiftingSupportLeftInstant.ERROR_TIME := T#10S;
	    "CylinderGeneratedCalls_DB".MM302_ShiftingSupportLeftInstant.ValveDelay := T#0ms;
	END_REGION
	
	REGION "CylinderGeneratedCalls_DB".MM304_MovingStopRightInstant
	    // Call Cylinder control "CylinderGeneratedCalls_DB".MM304_MovingStopRightInstantr
	    "CylinderGeneratedCalls_DB".MM304_MovingStopRightInstant.POWER_OK := true;
	    "CylinderGeneratedCalls_DB".MM304_MovingStopRightInstant.DELAY_BASIC := t#100ms;
	    "CylinderGeneratedCalls_DB".MM304_MovingStopRightInstant.DELAY_WORK := t#100ms;
	    "CylinderGeneratedCalls_DB".MM304_MovingStopRightInstant.DELAY_FREE := T#100mS;
	    "CylinderGeneratedCalls_DB".MM304_MovingStopRightInstant.ERROR_TIME := T#10S;
	    "CylinderGeneratedCalls_DB".MM304_MovingStopRightInstant.ValveDelay := T#0ms;
	END_REGION
	
	REGION "CylinderGeneratedCalls_DB".MM306_MovingStopLeftInstant
	    // Call Cylinder control "CylinderGeneratedCalls_DB".MM306_MovingStopLeftInstantr
	    "CylinderGeneratedCalls_DB".MM306_MovingStopLeftInstant.POWER_OK := true;
	    "CylinderGeneratedCalls_DB".MM306_MovingStopLeftInstant.DELAY_BASIC := t#100ms;
	    "CylinderGeneratedCalls_DB".MM306_MovingStopLeftInstant.DELAY_WORK := t#100ms;
	    "CylinderGeneratedCalls_DB".MM306_MovingStopLeftInstant.DELAY_FREE := T#100mS;
	    "CylinderGeneratedCalls_DB".MM306_MovingStopLeftInstant.ERROR_TIME := T#10S;
	    "CylinderGeneratedCalls_DB".MM306_MovingStopLeftInstant.ValveDelay := T#0ms;
	END_REGION
	
	REGION "CylinderGeneratedCalls_DB".MM340_RivetingUnitRightInstant
	    // Call Cylinder control "CylinderGeneratedCalls_DB".MM340_RivetingUnitRightInstantr
	    "CylinderGeneratedCalls_DB".MM340_RivetingUnitRightInstant.POWER_OK := true;
	    "CylinderGeneratedCalls_DB".MM340_RivetingUnitRightInstant.DELAY_BASIC := t#100ms;
	    "CylinderGeneratedCalls_DB".MM340_RivetingUnitRightInstant.DELAY_WORK := t#100ms;
	    "CylinderGeneratedCalls_DB".MM340_RivetingUnitRightInstant.DELAY_FREE := T#100mS;
	    "CylinderGeneratedCalls_DB".MM340_RivetingUnitRightInstant.ERROR_TIME := T#10S;
	    "CylinderGeneratedCalls_DB".MM340_RivetingUnitRightInstant.ValveDelay := T#0ms;
	END_REGION
	
	REGION "CylinderGeneratedCalls_DB".MM342_RivetingUnitLeftInstant
	    // Call Cylinder control "CylinderGeneratedCalls_DB".MM342_RivetingUnitLeftInstantr
	    "CylinderGeneratedCalls_DB".MM342_RivetingUnitLeftInstant.POWER_OK := true;
	    "CylinderGeneratedCalls_DB".MM342_RivetingUnitLeftInstant.DELAY_BASIC := t#100ms;
	    "CylinderGeneratedCalls_DB".MM342_RivetingUnitLeftInstant.DELAY_WORK := t#100ms;
	    "CylinderGeneratedCalls_DB".MM342_RivetingUnitLeftInstant.DELAY_FREE := T#100mS;
	    "CylinderGeneratedCalls_DB".MM342_RivetingUnitLeftInstant.ERROR_TIME := T#10S;
	    "CylinderGeneratedCalls_DB".MM342_RivetingUnitLeftInstant.ValveDelay := T#0ms;
	END_REGION
	
	REGION "CylinderGeneratedCalls_DB".MM344_RivetingSupportRightInstant
	    // Call Cylinder control "CylinderGeneratedCalls_DB".MM344_RivetingSupportRightInstantr
	    "CylinderGeneratedCalls_DB".MM344_RivetingSupportRightInstant.POWER_OK := true;
	    "CylinderGeneratedCalls_DB".MM344_RivetingSupportRightInstant.DELAY_BASIC := t#100ms;
	    "CylinderGeneratedCalls_DB".MM344_RivetingSupportRightInstant.DELAY_WORK := t#100ms;
	    "CylinderGeneratedCalls_DB".MM344_RivetingSupportRightInstant.DELAY_FREE := T#100mS;
	    "CylinderGeneratedCalls_DB".MM344_RivetingSupportRightInstant.ERROR_TIME := T#10S;
	    "CylinderGeneratedCalls_DB".MM344_RivetingSupportRightInstant.ValveDelay := T#0ms;
	END_REGION
	
	REGION "CylinderGeneratedCalls_DB".MM346_RivetingSupportLeftInstant
	    // Call Cylinder control "CylinderGeneratedCalls_DB".MM346_RivetingSupportLeftInstantr
	    "CylinderGeneratedCalls_DB".MM346_RivetingSupportLeftInstant.POWER_OK := true;
	    "CylinderGeneratedCalls_DB".MM346_RivetingSupportLeftInstant.DELAY_BASIC := t#100ms;
	    "CylinderGeneratedCalls_DB".MM346_RivetingSupportLeftInstant.DELAY_WORK := t#100ms;
	    "CylinderGeneratedCalls_DB".MM346_RivetingSupportLeftInstant.DELAY_FREE := T#100mS;
	    "CylinderGeneratedCalls_DB".MM346_RivetingSupportLeftInstant.ERROR_TIME := T#10S;
	    "CylinderGeneratedCalls_DB".MM346_RivetingSupportLeftInstant.ValveDelay := T#0ms;
	END_REGION
	
	REGION "CylinderGeneratedCalls_DB".MM350_ShiftWedgeRightInstant
	    // Call Cylinder control "CylinderGeneratedCalls_DB".MM350_ShiftWedgeRightInstantr
	    "CylinderGeneratedCalls_DB".MM350_ShiftWedgeRightInstant.POWER_OK := true;
	    "CylinderGeneratedCalls_DB".MM350_ShiftWedgeRightInstant.DELAY_BASIC := t#100ms;
	    "CylinderGeneratedCalls_DB".MM350_ShiftWedgeRightInstant.DELAY_WORK := t#100ms;
	    "CylinderGeneratedCalls_DB".MM350_ShiftWedgeRightInstant.DELAY_FREE := T#100mS;
	    "CylinderGeneratedCalls_DB".MM350_ShiftWedgeRightInstant.ERROR_TIME := T#10S;
	    "CylinderGeneratedCalls_DB".MM350_ShiftWedgeRightInstant.ValveDelay := T#0ms;
	END_REGION
	
	REGION "CylinderGeneratedCalls_DB".MM352_ShiftWedgeLeftInstant
	    // Call Cylinder control "CylinderGeneratedCalls_DB".MM352_ShiftWedgeLeftInstantr
	    "CylinderGeneratedCalls_DB".MM352_ShiftWedgeLeftInstant.POWER_OK := true;
	    "CylinderGeneratedCalls_DB".MM352_ShiftWedgeLeftInstant.DELAY_BASIC := t#100ms;
	    "CylinderGeneratedCalls_DB".MM352_ShiftWedgeLeftInstant.DELAY_WORK := t#100ms;
	    "CylinderGeneratedCalls_DB".MM352_ShiftWedgeLeftInstant.DELAY_FREE := T#100mS;
	    "CylinderGeneratedCalls_DB".MM352_ShiftWedgeLeftInstant.ERROR_TIME := T#10S;
	    "CylinderGeneratedCalls_DB".MM352_ShiftWedgeLeftInstant.ValveDelay := T#0ms;
	END_REGION
	
	REGION "CylinderGeneratedCalls_DB".MM104_AutoejectGripperLiftingInstant
	    // Call Cylinder control "CylinderGeneratedCalls_DB".MM104_AutoejectGripperLiftingInstantr
	    "CylinderGeneratedCalls_DB".MM104_AutoejectGripperLiftingInstant.POWER_OK := true;
	    "CylinderGeneratedCalls_DB".MM104_AutoejectGripperLiftingInstant.DELAY_BASIC := t#100ms;
	    "CylinderGeneratedCalls_DB".MM104_AutoejectGripperLiftingInstant.DELAY_WORK := t#100ms;
	    "CylinderGeneratedCalls_DB".MM104_AutoejectGripperLiftingInstant.DELAY_FREE := T#100mS;
	    "CylinderGeneratedCalls_DB".MM104_AutoejectGripperLiftingInstant.ERROR_TIME := T#10S;
	    "CylinderGeneratedCalls_DB".MM104_AutoejectGripperLiftingInstant.ValveDelay := T#0ms;
	END_REGION
	
	REGION "CylinderGeneratedCalls_DB".MM3100_SidememberSupportLeftInstant
	    // Call Cylinder control "CylinderGeneratedCalls_DB".MM3100_SidememberSupportLeftInstantr
	    "CylinderGeneratedCalls_DB".MM3100_SidememberSupportLeftInstant.POWER_OK := true;
	    "CylinderGeneratedCalls_DB".MM3100_SidememberSupportLeftInstant.DELAY_BASIC := t#100ms;
	    "CylinderGeneratedCalls_DB".MM3100_SidememberSupportLeftInstant.DELAY_WORK := t#100ms;
	    "CylinderGeneratedCalls_DB".MM3100_SidememberSupportLeftInstant.DELAY_FREE := T#100mS;
	    "CylinderGeneratedCalls_DB".MM3100_SidememberSupportLeftInstant.ERROR_TIME := T#10S;
	    "CylinderGeneratedCalls_DB".MM3100_SidememberSupportLeftInstant.ValveDelay := T#0ms;
	END_REGION
	
	REGION "CylinderGeneratedCalls_DB".MM3101_SidememberSupportRightInstant
	    // Call Cylinder control "CylinderGeneratedCalls_DB".MM3101_SidememberSupportRightInstantr
	    "CylinderGeneratedCalls_DB".MM3101_SidememberSupportRightInstant.POWER_OK := true;
	    "CylinderGeneratedCalls_DB".MM3101_SidememberSupportRightInstant.DELAY_BASIC := t#100ms;
	    "CylinderGeneratedCalls_DB".MM3101_SidememberSupportRightInstant.DELAY_WORK := t#100ms;
	    "CylinderGeneratedCalls_DB".MM3101_SidememberSupportRightInstant.DELAY_FREE := T#100mS;
	    "CylinderGeneratedCalls_DB".MM3101_SidememberSupportRightInstant.ERROR_TIME := T#10S;
	    "CylinderGeneratedCalls_DB".MM3101_SidememberSupportRightInstant.ValveDelay := T#0ms;
	END_REGION
	
	
	
	
END_FUNCTION

DATA_BLOCK "DB_Main_Instance"   // DB5000
VERSION : 0.1
// stored: AutoNumber false, DBAccessibleFromOPCUA true, DBAccessibleFromWebserver true, InstanceOfName FB_Main, InstanceOfType FB
"FB_Main"
BEGIN
   IEC_Timer_0_Instance.PT := T#0MS;
   IEC_Timer_0_Instance.IN := FALSE;
   F_TRIG_Instance.CLK := FALSE;
   F_TRIG_Instance.Q := FALSE;
   F_TRIG_Instance.Stat_Bit := FALSE;
   F_TRIG_Instance_1.CLK := FALSE;
   F_TRIG_Instance_1.Q := FALSE;
   F_TRIG_Instance_1.Stat_Bit := FALSE;
   F_TRIG_Instance_2.CLK := FALSE;
   F_TRIG_Instance_2.Q := FALSE;
   F_TRIG_Instance_2.Stat_Bit := FALSE;
   R_TRIG_Instance.CLK := FALSE;
   R_TRIG_Instance.Q := FALSE;
   R_TRIG_Instance.Stat_Bit := FALSE;
   R_TRIG_Instance_1.CLK := FALSE;
   R_TRIG_Instance_1.Q := FALSE;
   R_TRIG_Instance_1.Stat_Bit := FALSE;
END_DATA_BLOCK

DATA_BLOCK "Lamps_DB"   // DB25
VERSION : 0.1
// stored: AutoNumber true, DBAccessibleFromOPCUA true, DBAccessibleFromWebserver true, InstanceOfName Lamps, InstanceOfType FB
"Lamps"
BEGIN
   R_TRIG_Instance.CLK := FALSE;
   R_TRIG_Instance.Q := FALSE;
   R_TRIG_Instance.Stat_Bit := FALSE;
   IEC_Timer_0_Instance.PT := T#0MS;
   IEC_Timer_0_Instance.IN := FALSE;
END_DATA_BLOCK

DATA_BLOCK "ModeSelection_DB"   // DB56
VERSION : 0.1
// stored: AutoNumber true, DBAccessibleFromOPCUA true, DBAccessibleFromWebserver true, InstanceOfName ModeSelection, InstanceOfType FB
"ModeSelection"
BEGIN
   mode.activeMode := 1;
   mode.switch.auto := FALSE;
   mode.switch.poloautomaActivated := FALSE;
   mode.switch.stepModeActivated := FALSE;
   mode.button.basic.request.button := FALSE;
   mode.button.basic.request.visibility := FALSE;
   mode.button.auto.startRequest.button := FALSE;
   mode.button.auto.startRequest.visibility := FALSE;
   mode.button.auto.stopRequest.button := FALSE;
   mode.button.auto.stopRequest.visibility := FALSE;
   mode.button.auto.emptyRequest.button := FALSE;
   mode.button.auto.emptyRequest.visibility := FALSE;
   mode.button."step" := FALSE;
   mode.button.poloautomatStart[0..25] := FALSE;
   mode.modeChanged := FALSE;
   mode.autoStatus.stopping := FALSE;
   mode.autoStatus.stopped := FALSE;
   mode.autoStatus.emptying := FALSE;
   mode.autoStatus.empty := FALSE;
   mode.StationNrForPoloautomat_step := 0;
   F_TRIG_semiauto_switch.CLK := FALSE;
   F_TRIG_semiauto_switch.Q := FALSE;
   F_TRIG_semiauto_switch.Stat_Bit := FALSE;
   F_TRIG_switchAuto.CLK := FALSE;
   F_TRIG_switchAuto.Q := FALSE;
   F_TRIG_switchAuto.Stat_Bit := FALSE;
END_DATA_BLOCK

DATA_BLOCK "Default_SupervisionDB"   // DB68
VERSION : 0.1
// stored: AutoNumber true, DBAccessibleFromOPCUA true, DBAccessibleFromWebserver true, InstanceOfName Default_SupervisionFB, InstanceOfType FB
"Default_SupervisionFB"
   // VAR
   //    PC_Flags { ExternalWritable := 'False'; S7_SetPoint := 'True'} : PC_Flags_V2;
   //    State { ExternalWritable := 'False'; S7_SetPoint := 'True'} : SV_FB_State_V2;
   //    iOilHighLevekOK_O_1 { ExternalWritable := 'False'; S7_SetPoint := 'True'} : SV_State_V2;
   // END_VAR
BEGIN
END_DATA_BLOCK

DATA_BLOCK "AlarmsHandling_DB"   // DB16
VERSION : 0.1
// stored: AutoNumber true, DBAccessibleFromOPCUA true, DBAccessibleFromWebserver true, InstanceOfName AlarmsHandling, InstanceOfType FB
"AlarmsHandling"
   // VAR
   //    IEC_Timer_0_Instance_4 { S7_SetPoint := 'True'} : TON_TIME;
   //    IEC_Timer_0_Instance_5 { S7_SetPoint := 'True'} : TP_TIME;
   //    SetAlarmInstance { S7_SetPoint := 'True'} : Array[0..100] of "SetAlarm_PLC";
   //    AlarmPLCset { S7_SetPoint := 'True'} : Array[0..100] of Program_Alarm;
   // END_VAR
BEGIN
   IEC_Timer_0_Instance_4.PT := T#3S;
   IEC_Timer_0_Instance_4.IN := FALSE;
   IEC_Timer_0_Instance_5.PT := T#0MS;
   IEC_Timer_0_Instance_5.IN := FALSE;
   SetAlarmInstance[0..100].iAlarmCondition := FALSE;
   SetAlarmInstance[0..100].iReset := FALSE;
   SetAlarmInstance[0..14].iTime := T#0MS;
   SetAlarmInstance[15].iTime := T#8S;
   SetAlarmInstance[16..19].iTime := T#5S;
   SetAlarmInstance[20].iTime := T#0MS;
   SetAlarmInstance[21..24].iTime := T#5S;
   SetAlarmInstance[25].iTime := T#0MS;
   SetAlarmInstance[26..28].iTime := T#5S;
   SetAlarmInstance[29..100].iTime := T#0MS;
   SetAlarmInstance[0..100].AlarmToSet := FALSE;
   SetAlarmInstance[0..17].IEC_Timer_0_Instance.PT := T#0MS;
   SetAlarmInstance[18..19].IEC_Timer_0_Instance.PT := T#5S;
   SetAlarmInstance[20..100].IEC_Timer_0_Instance.PT := T#0MS;
   SetAlarmInstance[0..100].IEC_Timer_0_Instance.IN := FALSE;
   SetAlarmInstance[0..100].AlarmToSetWork := FALSE;
END_DATA_BLOCK

DATA_BLOCK "DB_DateTimeAndShifts_Instance"   // DB5010
VERSION : 0.1
// stored: AutoNumber false, DBAccessibleFromOPCUA true, DBAccessibleFromWebserver true, InstanceOfName FB_DateTimeAndShifts, InstanceOfType FB
"FB_DateTimeAndShifts"
BEGIN
   Settings.Actual.DateAndTime := DTL#2019-01-17-00:00:00;
   Settings.Actual.Shift1Enabled := TRUE;
   Settings.Actual.Shift1StartTime := TOD#06:00:00;
   Settings.Actual.Shift1EndTime := TOD#14:00:00;
   Settings.Actual.Shift2Enabled := TRUE;
   Settings.Actual.Shift2StartTime := TOD#14:00:00;
   Settings.Actual.Shift2EndTime := TOD#22:00:00;
   Settings.Actual.Shift3Enabled := TRUE;
   Settings.Actual.Shift3StartTime := TOD#22:00:00;
   Settings.Actual.Shift3EndTime := TOD#06:00:00;
   Settings.Last.DateAndTime := DTL#2019-01-17-00:00:00;
   Settings.Last.Shift1Enabled := TRUE;
   Settings.Last.Shift1StartTime := TOD#06:00:00;
   Settings.Last.Shift1EndTime := TOD#14:00:00;
   Settings.Last.Shift2Enabled := TRUE;
   Settings.Last.Shift2StartTime := TOD#14:00:00;
   Settings.Last.Shift2EndTime := TOD#22:00:00;
   Settings.Last.Shift3Enabled := TRUE;
   Settings.Last.Shift3StartTime := TOD#22:00:00;
   Settings.Last.Shift3EndTime := TOD#06:00:00;
   ShiftStatus.ShiftNumber := 1;
   ShiftStatus.ShiftActive := TRUE;
   ShiftStatus.Shift1Started := FALSE;
   ShiftStatus.Shift2Started := FALSE;
   ShiftStatus.Shift3Started := FALSE;
END_DATA_BLOCK

DATA_BLOCK "DB_Devices_Instance"   // DB5100
VERSION : 0.1
// stored: AutoNumber true, DBAccessibleFromOPCUA true, DBAccessibleFromWebserver true, InstanceOfName FB_Devices, InstanceOfType FB
"FB_Devices"
BEGIN
   ServiceDoors_Instance_1.iButtonOpen := FALSE;
   ServiceDoors_Instance_1.iButtonLock := FALSE;
   ServiceDoors_Instance_1.iSequenceStoped := TRUE;
   ServiceDoors_Instance_1.iSafetyOK := TRUE;
   ServiceDoors_Instance_1.iDoorClosed := TRUE;
   ServiceDoors_Instance_1.qStopSequence := FALSE;
   ServiceDoors_Instance_1.qUnlock := FALSE;
   ServiceDoors_Instance_1.qLightOpen := FALSE;
   ServiceDoors_Instance_1.qLightLock := FALSE;
   ServiceDoors_Instance_1.stopRequest := FALSE;
   ServiceDoors_Instance_2.iButtonOpen := FALSE;
   ServiceDoors_Instance_2.iButtonLock := FALSE;
   ServiceDoors_Instance_2.iSequenceStoped := TRUE;
   ServiceDoors_Instance_2.iSafetyOK := TRUE;
   ServiceDoors_Instance_2.iDoorClosed := TRUE;
   ServiceDoors_Instance_2.qStopSequence := FALSE;
   ServiceDoors_Instance_2.qUnlock := FALSE;
   ServiceDoors_Instance_2.qLightOpen := FALSE;
   ServiceDoors_Instance_2.qLightLock := FALSE;
   ServiceDoors_Instance_2.stopRequest := FALSE;
   R_TRIG_Instance.CLK := FALSE;
   R_TRIG_Instance.Q := FALSE;
   R_TRIG_Instance.Stat_Bit := FALSE;
   IEC_Timer_0_Instance.PT := T#0MS;
   IEC_Timer_0_Instance.IN := FALSE;
   IEC_Timer_0_Instance_1.PT := T#0MS;
   IEC_Timer_0_Instance_1.IN := FALSE;
   FB_TurnTable_Instance.iTurnTableInputs := 16#0000;
   FB_TurnTable_Instance.iPower := FALSE;
   FB_TurnTable_Instance.iSafety := FALSE;
   FB_TurnTable_Instance.iReset := FALSE;
   FB_TurnTable_Instance.iErrorReset := FALSE;
   FB_TurnTable_Instance.iManualMode := TRUE;
   FB_TurnTable_Instance.iAutomaticMode := FALSE;
   FB_TurnTable_Instance.iTurnTableInSafetyPosition := TRUE;
   FB_TurnTable_Instance.qTurnTableOutputs := 16#0000;
   FB_TurnTable_Instance.qeCommunication := FALSE;
   FB_TurnTable_Instance.qeTurnTablePosition := FALSE;
   FB_TurnTable_Instance.qeTurnTableSafetyPosition := FALSE;
   FB_TurnTable_Instance.qeTimeout := FALSE;
   FB_TurnTable_Instance.qePositionRunOver := FALSE;
   FB_TurnTable_Instance.qeSafety := FALSE;
   FB_TurnTable_Instance.qeSumError := FALSE;
   FB_TurnTable_Instance.qeSumWarning := FALSE;
   FB_TurnTable_Instance.Edges.Enabled := FALSE;
   FB_TurnTable_Instance.Edges.IndexerInPosition := TRUE;
   FB_TurnTable_Instance.TONs.tDelayCommunication.PT := T#0MS;
   FB_TurnTable_Instance.TONs.tDelayCommunication.IN := FALSE;
   FB_TurnTable_Instance.TONs.tDelayPositionError.PT := T#3S;
   FB_TurnTable_Instance.TONs.tDelayPositionError.IN := FALSE;
   FB_TurnTable_Instance.TONs.tDelayErrorReset.PT := T#0MS;
   FB_TurnTable_Instance.TONs.tDelayErrorReset.IN := FALSE;
   FB_TurnTable_Instance.RetentiveData.LastDirection := FALSE;
   FB_TurnTable_Instance.Commands.ReadyToJogCW := FALSE;
   FB_TurnTable_Instance.Commands.JogCW := FALSE;
   FB_TurnTable_Instance.Commands.ReadyToJogCCW := FALSE;
   FB_TurnTable_Instance.Commands.JogCCW := FALSE;
   FB_TurnTable_Instance.Commands.ReadyToStartCW := FALSE;
   FB_TurnTable_Instance.Commands.StartCW := FALSE;
   FB_TurnTable_Instance.Commands.ReadyToStartCCW := FALSE;
   FB_TurnTable_Instance.Commands.StartCCW := FALSE;
   F_TRIG_Instance.CLK := FALSE;
   F_TRIG_Instance.Q := FALSE;
   F_TRIG_Instance.Stat_Bit := FALSE;
   edges[1..6] := FALSE;
   R_TRIG_Instance_1.CLK := FALSE;
   R_TRIG_Instance_1.Q := FALSE;
   R_TRIG_Instance_1.Stat_Bit := FALSE;
   R_TRIG_Instance_2.CLK := FALSE;
   R_TRIG_Instance_2.Q := FALSE;
   R_TRIG_Instance_2.Stat_Bit := FALSE;
   R_TRIG_Instance_3.CLK := FALSE;
   R_TRIG_Instance_3.Q := FALSE;
   R_TRIG_Instance_3.Stat_Bit := FALSE;
   R_TRIG_Instance_4.CLK := FALSE;
   R_TRIG_Instance_4.Q := FALSE;
   R_TRIG_Instance_4.Stat_Bit := FALSE;
   R_TRIG_Instance_6.CLK := FALSE;
   R_TRIG_Instance_6.Q := FALSE;
   R_TRIG_Instance_6.Stat_Bit := FALSE;
   R_TRIG_Instance_7.CLK := FALSE;
   R_TRIG_Instance_7.Q := FALSE;
   R_TRIG_Instance_7.Stat_Bit := FALSE;
   R_TRIG_Instance_8.CLK := FALSE;
   R_TRIG_Instance_8.Q := FALSE;
   R_TRIG_Instance_8.Stat_Bit := FALSE;
   R_TRIG_Instance_5.CLK := FALSE;
   R_TRIG_Instance_5.Q := FALSE;
   R_TRIG_Instance_5.Stat_Bit := FALSE;
   edgesFitting[1..4] := FALSE;
   R_TRIG_V240Wp.CLK := FALSE;
   R_TRIG_V240Wp.Q := FALSE;
   R_TRIG_V240Wp.Stat_Bit := FALSE;
   R_TRIG_V240Bp.CLK := FALSE;
   R_TRIG_V240Bp.Q := FALSE;
   R_TRIG_V240Bp.Stat_Bit := FALSE;
   ReaderKeyence_Instance."I_address_Read Data 128Byte" := 697;
   ReaderKeyence_Instance."Q_address_Operation instruction Control Bits" := 699;
   ReaderKeyence_Instance."Q_address_Parameter Bank Number" := 701;
   ReaderKeyence_Instance.iReset := FALSE;
   ReaderKeyence_Instance.ResultData[1..128] := ' ';
   ReaderKeyence_Instance.ResultDataReadyCountOld := 0;
   ReaderKeyence_Instance.R_TRIG_Instance.CLK := FALSE;
   ReaderKeyence_Instance.R_TRIG_Instance.Q := FALSE;
   ReaderKeyence_Instance.R_TRIG_Instance.Stat_Bit := FALSE;
   ReaderKeyence_Instance.IEC_Timer_0_Instance.PT := T#0MS;
   ReaderKeyence_Instance.IEC_Timer_0_Instance.IN := FALSE;
   IEC_Timer_0_Instance_2.PT := T#0MS;
   IEC_Timer_0_Instance_2.IN := FALSE;
END_DATA_BLOCK

DATA_BLOCK "Manual_DB"   // DB53
VERSION : 0.1
// stored: AutoNumber true, DBAccessibleFromOPCUA true, DBAccessibleFromWebserver true, InstanceOfName Manual, InstanceOfType FB
"Manual"
   // VAR
   //    res : Bool := FALSE;
   //    R_TRIG_MM220bp { S7_SetPoint := 'True'} : R_TRIG;
   //    R_TRIG_MM220wp { S7_SetPoint := 'True'} : R_TRIG;
   //    R_TRIG_MM222bp { S7_SetPoint := 'True'} : R_TRIG;
   //    R_TRIG_MM222wp { S7_SetPoint := 'True'} : R_TRIG;
   //    R_TRIG_MM224bp { S7_SetPoint := 'True'} : R_TRIG;
   //    R_TRIG_MM224wp { S7_SetPoint := 'True'} : R_TRIG;
   // END_VAR
BEGIN
   R_TRIG_MM220bp.CLK := FALSE;
   R_TRIG_MM220bp.Q := FALSE;
   R_TRIG_MM220bp.Stat_Bit := FALSE;
   R_TRIG_MM220wp.CLK := FALSE;
   R_TRIG_MM220wp.Q := FALSE;
   R_TRIG_MM220wp.Stat_Bit := FALSE;
   R_TRIG_MM222bp.CLK := FALSE;
   R_TRIG_MM222bp.Q := FALSE;
   R_TRIG_MM222bp.Stat_Bit := FALSE;
   R_TRIG_MM222wp.CLK := FALSE;
   R_TRIG_MM222wp.Q := FALSE;
   R_TRIG_MM222wp.Stat_Bit := FALSE;
   R_TRIG_MM224bp.CLK := FALSE;
   R_TRIG_MM224bp.Q := FALSE;
   R_TRIG_MM224bp.Stat_Bit := FALSE;
   R_TRIG_MM224wp.CLK := FALSE;
   R_TRIG_MM224wp.Q := FALSE;
   R_TRIG_MM224wp.Stat_Bit := FALSE;
END_DATA_BLOCK

DATA_BLOCK "DB_Eks_Instance"   // DB5050
VERSION : 0.1
// stored: AutoNumber false, DBAccessibleFromOPCUA true, DBAccessibleFromWebserver true, InstanceOfName FB_Eks, InstanceOfType FB
"FB_Eks"
BEGIN
   KeyInsertedInReader.CLK := TRUE;
   KeyInsertedInReader.Q := FALSE;
   KeyInsertedInReader.Stat_Bit := TRUE;
   KeyRemovedFromReader.CLK := TRUE;
   KeyRemovedFromReader.Q := FALSE;
   KeyRemovedFromReader.Stat_Bit := TRUE;
   TONs.tDelayTimeoutError.PT := T#0MS;
   TONs.tDelayTimeoutError.IN := FALSE;
END_DATA_BLOCK

